IF bError THEN
	eCurrentState := E_MachineState.MACHINESTATE_Error;
	bBusy := FALSE;
	aPumps[nPumpNrRinsePump].M_Off();
	aPumps[nPumpNrWastePump].M_Off();
END_IF

//Prozessdaten aktualisieren
stProcessData.nObjId := nObjectID;
stProcessData.n32Data[0] := BOOL_TO_DINT(bIsInit);
stProcessData.n32Data[1] := eCurrentState;
stProcessData.n32Data[2] := stError.ErrorId;

stProcessData.n32Data[3] := BOOL_TO_DINT(bRinse);

stProcessData.n32Data[4] := BOOL_TO_DINT(aPumps[nPumpNrWastePump].P_bIsOn);
aObjProcData[nNotifyId] := stProcessData;

ACTION A_EmptyWaste:
IF nStateA_EmptyWaste = 0 THEN	//Wastepumpe einschalten
	aPumps[nPumpNrWastePump].M_On();
	tmrEmptyFluid(IN:= TRUE, PT:= T#10S);
	nStateA_EmptyWaste := 1;
ELSIF nStateA_EmptyWaste = 1 THEN //Warten auf Timer und Wastepumpe ausschalten
	tmrEmptyFluid();
	IF tmrEmptyFluid.Q THEN
		tmrEmptyFluid(IN:= FALSE);
		aPumps[nPumpNrWastePump].M_Off();
		IF NOT bLevelSensor THEN	//Leeren
			IF nPumpNrRinsePump > 0 THEN
				aPumps[nPumpNrRinsePump].M_Off();	
			END_IF
			stError.ErrorId := E_ErrorIdCmd.ERRORID_TimeOut;
			stError.POUState := nStateA_EmptyWaste;
			nStateA_EmptyWaste := 99;
		END_IF
		nStateA_EmptyWaste := 80;
	END_IF
ELSIF nStateA_EmptyWaste = 70 THEN
	tmrEmptyFluid(IN:= FALSE);
	nStateA_EmptyWaste := 80;
END_IF

//Errorhandling
IF nStateA_EmptyWaste = 99 THEN
	stError.Cmd := E_Action.ACTION_EmptyWaste;
	stError.POUAction := E_POUACT.POUACT_A_EmptyWaste;
	fbErrorList.M_Add(stError);
END_IF
END_ACTION

ACTION A_Rinse:
//Überwachung des Wastebottles
stError.ErrorId := M_CheckBottles();
IF stError.ErrorId > 0 THEN
	stError.POUState := nStateA_Rinse;
	nStateA_Rinse := 99;
END_IF

CASE nStateA_Rinse OF
	0:	IF bRinseOn THEN
			//WastePump EIN
			//RinsePump EIN
			aPumps[nPumpNrWastePump].M_On();
			aPumps[nPumpNrRinsePump].P_nStartSpeed := aStRinseChannels[nRinseChannel].nStartSpeed;
			aPumps[nPumpNrRinsePump].P_nRatedSpeed := aStRinseChannels[nRinseChannel].nRatedSpeed;
			aPumps[nPumpNrRinsePump].P_nDelay := aStRinseChannels[nRinseChannel].nStartTime;
			IF aStRinseChannels[nRinseChannel].nValveNr > 0 THEN
				aValves[aStRinseChannels[nRinseChannel].nValveNr].M_On(1);
			END_IF
			
			IF aPumps[nPumpNrRinsePump].M_On() THEN
				IF tmrRinse.PT > T#0MS THEN
					tmrRinse.IN := TRUE;
					nStateA_Rinse := 1;
				ELSE
					nStateA_Rinse := 1;
				END_IF
			END_IF
		ELSE
			bEmptyWaste := TRUE;
			M_RinsePumpOff();
			nStateA_Rinse := 80;
		END_IF

	1:	//Rinse aktiv (Überwachung des LevelSensors und des Rinse-Timers
		tmrRinse();
		IF bRinseOn THEN
			IF tmrRinse.Q THEN
				nStateA_Rinse := 3;
				RETURN;	
			END_IF
		
			IF NOT bLevelSensor THEN	//RinsePumpe für 2s "AUS" und dann wieder "EIN"
				M_RinsePumpOff();
				tmrRinsePause(IN:= TRUE, PT:= T#2S);
				nStateA_Rinse := 2;
			END_IF
		ELSE
			tmrRinsePause(IN:= FALSE);
			nStateA_Rinse := 3;
		END_IF
		
	2:	//Warten bis Timer abgelaufen
		IF bRinseOn THEN
			tmrRinse();
			IF tmrRinse.Q THEN
				tmrRinsePause(IN:= FALSE);
				//Hier sollte der Sensor spätestens wieder frei sein
				IF NOT bLevelSensor THEN
					stError.ErrorId := E_ErrorIdCmd.ERRORID_TimeOut;
					stError.POUState := nStateA_Rinse;
					nStateA_Rinse := 99; //Error
				ELSE
					nStateA_Rinse := 0; //Pumpe wieder einschalten??	
				END_IF
			END_IF
		ELSE
			tmrRinse(IN:= FALSE);
			nStateA_Rinse := 3;
		END_IF
		
	3:	//Aus
		tmrRinse(IN:=FALSE);
		IF NOT bKeepWastePumpOn THEN
			bEmptyWaste := TRUE;
		END_IF
		M_RinsePumpOff();
		nStateA_Rinse := 80;
		
	70:	//Abbrechen
		aPumps[nPumpNrWastePump].M_Off();
		M_RinsePumpOff();

		tmrRinse(IN:= FALSE);
		nStateA_Rinse := 80;

	90: //Error - Abbrechen
		aPumps[nPumpNrWastePump].M_Off();
		M_RinsePumpOff();
		tmrRinse(IN:= FALSE);
		tmrRinsePause(IN:= FALSE);
END_CASE

//Errorhandling
IF nStateA_Rinse = 99 THEN
	aPumps[nPumpNrWastePump].M_Off();
	M_RinsePumpOff();
	tmrRinse(IN:= FALSE);
	tmrRinsePause(IN:= FALSE);
	stError.Cmd := E_Action.ACTION_Rinse;
	stError.POUAction := E_POUACT.POUACT_A_Rinse;
	fbErrorList.M_Add(stError);
END_IF
END_ACTION

ACTION A_SwitchPump:
IF nStateA_SwitchPump = 0 THEN
	//Welche Pumpe soll geschalten werden?
	//0= Waste
	//>0 = RinseChannel
	IF nSwitchChannel = 0 THEN
		IF bSwitchOn THEN	//Waste-Pumpe einschalten
			//Falls EmptyWaste noch aktiv ist, dieses abbrechen, da EmptyWaste die Pumpe wieder abschaltet
			M_CancelAction(E_Action.ACTION_EmptyWaste);
			aPumps[nPumpNrWastePump].M_On();
		ELSE	//Ausschalten
			aPumps[nPumpNrWastePump].M_Off();
		END_IF
		nStateA_SwitchPump := 80;
	ELSIF nSwitchChannel > 0 THEN
		IF bSwitchOn THEN	//Einschalten
			aPumps[nPumpNrRinsePump].P_nStartSpeed := aStRinseChannels[nRinseChannel].nStartSpeed;
			aPumps[nPumpNrRinsePump].P_nRatedSpeed := aStRinseChannels[nRinseChannel].nRatedSpeed;
			aPumps[nPumpNrRinsePump].P_nDelay := aStRinseChannels[nRinseChannel].nStartTime;
			IF aStRinseChannels[nRinseChannel].nValveNr > 0 THEN
				aValves[aStRinseChannels[nRinseChannel].nValveNr].M_On(1);
			END_IF				
		ELSE	//Ausschalten
			M_RinsePumpOff();
		END_IF
			nStateA_SwitchPump := 80;
	END_IF
ELSIF nStateA_SwitchPump = 70 THEN
	aPumps[nPumpNrWastePump].M_Off();
	M_RinsePumpOff();
	nStateA_SwitchPump := 80;
END_IF
END_ACTION

METHOD FB_init : BOOL
VAR_INPUT
	bInitRetains : BOOL; // if TRUE, the retain variables are initialized (warm start / cold start)
	bInCopyCode : BOOL;  // if TRUE, the instance afterwards gets moved into the copy code (online change)
END_VAR
eObjectType := E_ObjectType.OBJECTTYPE_WashStation;
eObjectGroup := E_ObjectGroup.OBJECTGROUP_Target OR E_ObjectGroup.OBJECTGROUP_Device;
END_METHOD

METHOD M_ApplyPos : ERRORID
VAR_INPUT
	eTargetRef 		: E_TargetRef;
	nPointSlotNr	: UINT;
	stPos 			: ST_3DPoint;
	bXPos			: BOOL;
	bYPos			: BOOL;
	bZPos			: BOOL;	
END_VAR

VAR
	stAbsPos		: ST_3DPoint;
END_VAR
IF eTargetRef = E_TargetRef.TARGETREF_SpecPoint THEN
	stAbsPos := P_stAbsPosLB;
	IF bXPos THEN
		aStWashPoints[nPointSlotNr].X := stPos.X - stAbsPos.X;
	END_IF
	IF bYPos THEN
		aStWashPoints[nPointSlotNr].Y := stPos.Y - stAbsPos.Y;
	END_IF
	IF bZPos THEN
		aStWashPoints[nPointSlotNr].Z := stPos.Z - stAbsPos.Z;
	END_IF		
ELSE
	M_ApplyPos := SUPER^.M_ApplyPos(eTargetRef, nPointSlotNr, stPos,bXPos, bYPos, bZPos);	
END_IF
END_METHOD

METHOD M_CancelAction
VAR_INPUT
	eAction : E_Action;
END_VAR
CASE eAction OF
	E_Action.ACTION_Rinse:
		IF bRinse AND nStateA_Rinse < 70 THEN
			nStateA_Rinse := 70;
		END_IF
	E_Action.ACTION_SwitchPump:
		IF bSwitchPump AND nStateA_SwitchPump < 70 THEN
			nStateA_SwitchPump := 70;
		END_IF
	E_Action.ACTION_EmptyWaste:
		IF bEmptyWaste AND nStateA_EmptyWaste < 70 THEN
			nStateA_EmptyWaste := 70;
		END_IF
END_CASE
END_METHOD

METHOD M_CheckAction : ERRORID
VAR_INPUT
	refActionData 	: REFERENCE TO ST_ActionData;
	pCorrelObject	: POINTER TO FB_Object;
END_VAR
IF refActionData.eAction = E_Action.ACTION_TeachTarget THEN
	IF NOT DINT_TO_UINT(refActionData.aParams[1]) = E_TargetRef.TARGETREF_SpecPoint AND (refActionData.aParams[2] = 1 AND refActionData.aParams[2] = 2) THEN
		M_CheckAction := E_ErrorIdCmd.ERRORID_InvalidTargetPointRef;
	END_IF
ELSIF refActionData.eAction = E_Action.ACTION_WashTool THEN
	//SpecPoint prüfen
	IF NOT (refActionData.aParams[1] > 0 AND refActionData.aParams[1] <= nNoOfWashPoints) THEN
		M_CheckAction := E_ErrorIdCmd.ERRORID_InvalidTargetPointNr;
		RETURN;
	END_IF
	//Washmode prüfen
	IF NOT(refActionData.aParams[2] = E_WashMode.MODE_WashInside OR
		refActionData.aParams[2] = E_WashMode.MODE_WashOutside OR
		refActionData.aParams[2] = E_WashMode.MODE_WashInOutside OR
		refActionData.aParams[2] = E_WashMode.MODE_DryOutside) THEN
		M_CheckAction := E_ErrorIdCmd.ERRORID_InvalidWashMode;
		RETURN;
	END_IF
	//BottleState prüfen
	M_CheckAction := M_CheckBottles();
END_IF
END_METHOD

METHOD M_CheckBottles : ERRORID
VAR_INPUT
END_VAR
//Systemliquidbottle OK?
IF nSysLiquidBottle > 0 THEN
	IF NOT aSensSysLiquidBottle[nSysLiquidBottle] THEN //Leer
		M_CheckBottles := E_ErrorIdCmd.ERRORID_LiquidBottleEmpty;
		RETURN;
	END_IF
END_IF
//Wastebottle OK?
IF nWasteBottle > 0 THEN
	IF NOT aSensWasteBottle[nWasteBottle] THEN //Voll
		M_CheckBottles := E_ErrorIdCmd.ERRORID_WasteBottleFull;
		RETURN;
	END_IF
END_IF
END_METHOD

METHOD M_CheckProcDataType : BOOL
VAR_INPUT
	eProcDataType : E_ProcDataType;
END_VAR
END_METHOD

METHOD M_ExeAction : ERRORID
VAR_INPUT
	refActionData : REFERENCE TO ST_ActionData;	
END_VAR
IF refActionData.eAction = E_Action.ACTION_Init THEN
	bIsInit := TRUE;
	RETURN;
ELSIF refActionData.eAction = E_Action.ACTION_SwitchPump THEN
	IF NOT bSwitchPump THEN
		nSwitchChannel := DINT_TO_USINT(refActionData.aParams[1]);
		IF NOT(nSwitchChannel >= 0 AND nSwitchChannel <= nNoOfRinseChannels) THEN
			M_ExeAction := E_ErrorIdCmd.ERRORID_InvalidPumpNr;
			RETURN;			
		END_IF
		bSwitchOn := DINT_TO_BOOL(refActionData.aParams[2]);
		bSwitchPump := TRUE;
	ELSE
		RETURN;
	END_IF
	
ELSIF refActionData.eAction = E_Action.ACTION_EmptyWaste THEN
	IF NOT aSensWasteBottle[nWasteBottle] THEN
		M_ExeAction := E_ErrorIdCmd.ERRORID_WasteBottleFull;
		RETURN;
	END_IF
	IF NOT bEmptyWaste THEN
		bEmptyWaste := TRUE;
	ELSE
		RETURN;
	END_IF

ELSIF refActionData.eAction = E_Action.ACTION_Stop THEN
	IF bRinse THEN
		bRinseOn := FALSE;
	ELSE
		aPumps[nPumpNrWastePump].M_Off();
		M_RinsePumpOff();
	END_IF	
	
ELSIF refActionData.eAction = E_Action.ACTION_Rinse THEN
	nRinseChannel := DINT_TO_USINT(refActionData.aParams[1]);
	tmrRinse.PT := DINT_TO_TIME(refActionData.aParams[3]);
	IF NOT(nRinseChannel >= 1 AND nRinseChannel <= nNoOfRinseChannels) THEN
		M_ExeAction := E_ErrorIdCmd.ERRORID_InvalidRinseChannel;
		RETURN;
	END_IF
	nPumpNrRinsePump := aStRinseChannels[nRinseChannel].nPumpNr;
	bRinseOn := DINT_TO_BOOL(refActionData.aParams[2]);
	bKeepWastePumpOn := DINT_TO_BOOL(refActionData.aParams[4]);
	bRinse := TRUE;
ELSE
	M_ExeAction := E_ErrorIdCmd.ERRORID_InvalidAction;
	RETURN;
END_IF
bBusy := TRUE;
eCurrentState:= E_MachineState.MACHINESTATE_Active;
END_METHOD

METHOD M_GetAbsPos : ST_3DPoint
VAR_INPUT
	pChildPos	: POINTER TO ST_3DPoint;
	eTargetRef 	: E_TargetRef;
	nParam1		: UINT;
 	nParam2		: UINT;
	nParam3		: USINT;
	nParam4		: USINT;
	nZLevel		: USINT;
END_VAR
VAR_OUTPUT
	nErrorId 	: ERRORID;
	lrAngle		: LREAL;
END_VAR
VAR
	stLocPosLB : ST_3DPoint;
END_VAR
IF eTargetRef = E_TargetRef.TARGETREF_SpecPoint THEN
	IF nParam1 > 0 AND nParam1 <= cMaxWashPoints THEN
		stLocPosLB := P_stRelPosLB;
		stLocPosLB := F_Add3DPoints(stLocPosLB,aStWashPoints[nParam1]);
		M_GetAbsPos := pParentTarget^.M_GetAbsPos(pChildPos := ADR(stLocPosLB), eTargetRef:= E_TargetRef.TARGETREF_LeftBottom,
														nParam1:= 0,
														nParam2:= 0, nParam3:= 0,nParam4:= 0, nZLevel:= 0,
														lrAngle => lrAngle, nErrorId=> nErrorId);		
	ELSE
		nErrorId := E_ErrorIdCmd.ERRORID_InvalidTargetPointNr;
	END_IF
ELSE
	M_GetAbsPos := SUPER^.M_GetAbsPos(pChildPos := pChildPos, eTargetRef:= eTargetRef,
													nParam1:= nParam1,
													nParam2:= nParam2, nParam3:= nParam3, nParam4:= 0, nZLevel:= nZLevel,
													lrAngle => lrAngle, nErrorId=> nErrorId);	
END_IF
END_METHOD

METHOD M_GetActionBusy : BOOL
VAR_INPUT
	eAction : E_Action;
END_VAR
IF eAction = E_Action.ACTION_SwitchPump THEN
	M_GetActionBusy := bSwitchPump;
ELSIF eAction = E_Action.ACTION_EmptyWaste THEN
	M_GetActionBusy := bEmptyWaste;
ELSIF eAction = E_Action.ACTION_Rinse THEN
	M_GetActionBusy := bRinse;
END_IF
END_METHOD

METHOD M_GetAllProps : ERRORID
VAR_INPUT
	refCmdData : REFERENCE TO  ST_CmdData;
END_VAR

VAR
	i : USINT;
END_VAR
SUPER^.M_GetAllProps(refCmdData); 

//RinseChannels
nCurrentPropIndex := nCurrentPropIndex + 1;
refCmdData.n32Data[nCurrentPropIndex] := nNoOfRinseChannels;
//In Abhängigkeit von der Anzahl der RinseChannels , diese aus RinseChannel-Array lesen
FOR i:= 1 TO nNoOfRinseChannels BY 1 DO
	nCurrentPropIndex := nCurrentPropIndex + 1;	//PumpNr
	refCmdData.n32Data[nCurrentPropIndex] := aStRinseChannels[i].nPumpNr;
	nCurrentPropIndex := nCurrentPropIndex + 1;	//ValveNr
	refCmdData.n32Data[nCurrentPropIndex] := aStRinseChannels[i].nValveNr;
	nCurrentPropIndex := nCurrentPropIndex + 1;	//StartSpeed in %
	refCmdData.n32Data[nCurrentPropIndex] := aStRinseChannels[i].nStartSpeed;
	nCurrentPropIndex := nCurrentPropIndex + 1;	//RatedSpeed in %
	refCmdData.n32Data[nCurrentPropIndex] := aStRinseChannels[i].nRatedSpeed;
	nCurrentPropIndex := nCurrentPropIndex + 1;	//StartTime in ms
	refCmdData.n32Data[nCurrentPropIndex] := aStRinseChannels[i].nStartTime;
END_FOR

//WashPoints
nCurrentPropIndex := nCurrentPropIndex + 1;
refCmdData.n32Data[nCurrentPropIndex] := nNoOfWashPoints; 
//In Abhängigkeit von der Anzahl der Waschpunkte , diese aus WashPoint-Array lesen
FOR i:= 1 TO nNoOfWashPoints BY 1 DO
	nCurrentPropIndex := nCurrentPropIndex + 1;
	refCmdData.n32Data[nCurrentPropIndex] := REAL_TO_DINT(aStWashPoints[i].X);
	nCurrentPropIndex := nCurrentPropIndex + 1;
	refCmdData.n32Data[nCurrentPropIndex] := REAL_TO_DINT(aStWashPoints[i].Y);
	nCurrentPropIndex := nCurrentPropIndex + 1;
	refCmdData.n32Data[nCurrentPropIndex] := REAL_TO_DINT(aStWashPoints[i].Z);
	nCurrentPropIndex := nCurrentPropIndex + 1;
	refCmdData.n32Data[nCurrentPropIndex] := REAL_TO_DINT(aStWashPoints[i].nRinseChannel);
END_FOR

nCurrentPropIndex := nCurrentPropIndex + 1;
refCmdData.n32Data[nCurrentPropIndex] := nPumpNrWastePump;
nCurrentPropIndex := nCurrentPropIndex + 1;
refCmdData.n32Data[nCurrentPropIndex] := nSysLiquidBottle;
nCurrentPropIndex := nCurrentPropIndex + 1;
refCmdData.n32Data[nCurrentPropIndex] := nWasteBottle;
nCurrentPropIndex := nCurrentPropIndex + 1;
refCmdData.n32Data[nCurrentPropIndex] := nValveNrAirShower;
nCurrentPropIndex := nCurrentPropIndex + 1;
refCmdData.n32Data[nCurrentPropIndex] := nGCodeTargetNr;
END_METHOD

METHOD M_GetProcData : DINT
VAR_INPUT
	eProcDataType : E_ProcDataType;
END_VAR
END_METHOD

METHOD M_GetRinseChannel : USINT
VAR_INPUT
	nWashPointNr : USINT;
END_VAR
IF nWashPointNr > 0 AND nWashPointNr <= nNoOfWashPoints THEN
	M_GetRinseChannel := aStWashPoints[nWashPointNr].nRinseChannel;
END_IF
END_METHOD

METHOD M_Reset
bError := FALSE;
bBusy := FALSE;
eCurrentState := E_MachineState.MACHINESTATE_Idle;
END_METHOD

METHOD PRIVATE M_RinsePumpOff
VAR_INPUT
END_VAR

VAR
	i		: USINT;
	nTemp 	: USINT;
END_VAR
FOR i := 1 TO nNoOfRinseChannels BY 1 DO
	nTemp := aStRinseChannels[i].nPumpNr;
	IF nTemp > 0 THEN
		aPumps[nTemp].M_Off();
	END_IF
	nTemp := aStRinseChannels[i].nValveNr;
	IF nTemp > 0 THEN
		aValves[nTemp].M_Off();
	END_IF
END_FOR
END_METHOD

METHOD M_SetAllProps : ERRORID
VAR_INPUT
	refCmdData : REFERENCE TO  ST_CmdData;
END_VAR

VAR
	i : USINT;
END_VAR
M_SetAllProps := SUPER^.M_SetAllProps(refCmdData);

IF M_SetAllProps > 0 THEN
	RETURN;
END_IF

//RinseChannels
nCurrentPropIndex := nCurrentPropIndex + 1;
nSpecPropIndex := nCurrentPropIndex;
nNoOfRinseChannels := DINT_TO_USINT(refCmdData.n32Data[nCurrentPropIndex]); 
//In Abhängigkeit von der Anzahl der RinseChannels , diese in RinseChannel-Array schreiben
IF NOT (nNoOfRinseChannels > 0 AND nNoOfRinseChannels <= cMaxRinseChannels) THEN
	M_SetAllProps := E_ErrorIdObjMgmt.ERRORID_InvalidNoOfRinseChannels;
	RETURN;
END_IF

FOR i:= 1 TO nNoOfRinseChannels BY 1 DO
	nCurrentPropIndex := nCurrentPropIndex + 1; //PumpNr
	IF refCmdData.n32Data[nCurrentPropIndex] >= 0 AND refCmdData.n32Data[nCurrentPropIndex] <= cNoOfPumps THEN
		aStRinseChannels[i].nPumpNr := DINT_TO_USINT(refCmdData.n32Data[nCurrentPropIndex]);
	ELSE
		M_SetAllProps := E_ErrorIdCmd.ERRORID_InvalidPumpNr;
		RETURN;
	END_IF
	nCurrentPropIndex := nCurrentPropIndex + 1;	//ValveNr
	IF refCmdData.n32Data[nCurrentPropIndex] >= 0 AND refCmdData.n32Data[nCurrentPropIndex] <= cNoOfValves THEN
		aStRinseChannels[i].nValveNr := DINT_TO_USINT(refCmdData.n32Data[nCurrentPropIndex]);
	ELSE
		M_SetAllProps := E_ErrorIdObjMgmt.ERRORID_InvalidValveNumber;
		RETURN;
	END_IF
	nCurrentPropIndex := nCurrentPropIndex + 1;	//StartSpeed in %
	aStRinseChannels[i].nStartSpeed := DINT_TO_USINT(refCmdData.n32Data[nCurrentPropIndex]);
	nCurrentPropIndex := nCurrentPropIndex + 1;	//RatedSpeed in %
	aStRinseChannels[i].nRatedSpeed := DINT_TO_USINT(refCmdData.n32Data[nCurrentPropIndex]);
	nCurrentPropIndex := nCurrentPropIndex + 1;	//StartTime in ms
	aStRinseChannels[i].nStartTime := DINT_TO_UINT(refCmdData.n32Data[nCurrentPropIndex]);
END_FOR

//WashPoints
nCurrentPropIndex := nCurrentPropIndex + 1;
nNoOfWashPoints := DINT_TO_USINT(refCmdData.n32Data[nCurrentPropIndex]); 
//In Abhängigkeit von der Anzahl der Waschpunkte , diese in WashPoint-Array schreiben
IF NOT (nNoOfWashPoints > 0 AND nNoOfWashPoints <= cMaxWashPoints) THEN
	M_SetAllProps := E_ErrorIdObjMgmt.ERRORID_InvalidNoOfSpecPoints;
	RETURN;
END_IF

FOR i:= 1 TO nNoOfWashPoints BY 1 DO
	nCurrentPropIndex := nCurrentPropIndex + 1;
	aStWashPoints[i].X := DINT_TO_REAL(refCmdData.n32Data[nCurrentPropIndex]);
	nCurrentPropIndex := nCurrentPropIndex + 1;
	aStWashPoints[i].Y := DINT_TO_REAL(refCmdData.n32Data[nCurrentPropIndex]);
	nCurrentPropIndex := nCurrentPropIndex + 1;
	aStWashPoints[i].Z := DINT_TO_REAL(refCmdData.n32Data[nCurrentPropIndex]);
	nCurrentPropIndex := nCurrentPropIndex + 1;
	//Zugeordneter RinseChannel
	aStWashPoints[i].nRinseChannel := DINT_TO_USINT(refCmdData.n32Data[nCurrentPropIndex]);;
END_FOR

//WastePump
nCurrentPropIndex := nCurrentPropIndex + 1;
IF refCmdData.n32Data[nCurrentPropIndex] >= 1 AND refCmdData.n32Data[nCurrentPropIndex] <= cNoOfPumps THEN
	nPumpNrWastePump := DINT_TO_USINT(refCmdData.n32Data[nCurrentPropIndex]);
ELSE
	M_SetAllProps := E_ErrorIdCmd.ERRORID_InvalidPumpNr;
END_IF

//LiquidBottle
nCurrentPropIndex := nCurrentPropIndex + 1;
IF refCmdData.n32Data[nCurrentPropIndex] >= 1 AND refCmdData.n32Data[nCurrentPropIndex] <= cNoOfLiquidBottles THEN
	nSysLiquidBottle := DINT_TO_USINT(refCmdData.n32Data[nCurrentPropIndex]);
ELSE
	M_SetAllProps := E_ErrorIdObjMgmt.ERRORID_InvalidLiquidbottle;
END_IF

//WasteBottle
nCurrentPropIndex := nCurrentPropIndex + 1;
IF refCmdData.n32Data[nCurrentPropIndex] >= 1 AND refCmdData.n32Data[nCurrentPropIndex] <= cNoOfWasteBottles THEN
	nWasteBottle := DINT_TO_USINT(refCmdData.n32Data[nCurrentPropIndex]);
ELSE
	M_SetAllProps := E_ErrorIdObjMgmt.ERRORID_InvalidWastebottle;
END_IF

//ValveNrDrying (Trockendusche für pH Elektrode)
nCurrentPropIndex := nCurrentPropIndex + 1;
IF refCmdData.n32Data[nCurrentPropIndex] >= 0 AND refCmdData.n32Data[nCurrentPropIndex] <= cNoOfValves THEN
	nValveNrAirShower := DINT_TO_USINT(refCmdData.n32Data[nCurrentPropIndex]);
ELSE
	M_SetAllProps := E_ErrorIdObjMgmt.ERRORID_InvalidValveNumber;
END_IF
nCurrentPropIndex := nCurrentPropIndex + 1;
nGCodeTargetNr := DINT_TO_UINT(refCmdData.n32Data[nCurrentPropIndex]);
nNoOfProps := nCurrentPropIndex + 1;
END_METHOD

METHOD M_SetSingleProp : ERRORID
VAR_INPUT
	refCmdData : REFERENCE TO  ST_CmdData;
END_VAR

VAR
	i : UINT;
	nIndex					: UINT;
	nIndexRinseChannels	 	: UINT;
	nIndexWashPoints 	 	: UINT;
	nIndexRestProps 	 	: UINT;
END_VAR
nIndexRinseChannels := nSpecPropIndex;
nIndexWashPoints := nIndexRinseChannels + nNoOfRinseChannels * 5 + 1;
nIndexRestProps := nIndexWashPoints + nNoOfWashPoints * 4 + 1;

//Section: RinseChannels
IF refCmdData.aHeader[1] > nIndexRinseChannels AND refCmdData.aHeader[1] < nIndexWashPoints THEN
	FOR i:= 1 TO nNoOfRinseChannels BY 1 DO
		//ersten Index innerhalb der Section ermitteln
		nIndex := nIndexRinseChannels + ((i - 1) * 5) + 1;
		IF refCmdData.aHeader[1] = nIndex THEN	//PumpNr
			IF refCmdData.n32Data[0] >= 0 AND refCmdData.n32Data[0] <= cNoOfPumps THEN
				aStRinseChannels[i].nPumpNr := DINT_TO_USINT(refCmdData.n32Data[0]);
			ELSE
				M_SetSingleProp := E_ErrorIdCmd.ERRORID_InvalidPumpNr;
				RETURN;
			END_IF
			RETURN;
		ELSIF refCmdData.aHeader[1] = nIndex + 1 THEN	//ValveNr
			IF refCmdData.n32Data[0] >= 0 AND refCmdData.n32Data[0] <= cNoOfValves THEN
				aStRinseChannels[i].nValveNr := DINT_TO_USINT(refCmdData.n32Data[0]);
			ELSE
				M_SetSingleProp := E_ErrorIdObjMgmt.ERRORID_InvalidValveNumber;
				RETURN;
			END_IF
		ELSIF refCmdData.aHeader[1] = nIndex + 2 THEN	//StartSpeed in %
			aStRinseChannels[i].nStartSpeed := DINT_TO_USINT(refCmdData.n32Data[0]);	
		ELSIF refCmdData.aHeader[1] = nIndex + 3 THEN	//RatedSpeed in %
			aStRinseChannels[i].nRatedSpeed := DINT_TO_USINT(refCmdData.n32Data[0]);
		ELSIF refCmdData.aHeader[1] = nIndex + 4 THEN	//StartTime in ms
			aStRinseChannels[i].nStartTime := DINT_TO_UINT(refCmdData.n32Data[0]);
		END_IF		
	END_FOR
//Section: Washpoints	
ELSIF refCmdData.aHeader[1] > nIndexWashPoints AND refCmdData.aHeader[1] < nIndexRestProps THEN
	FOR i:= 1 TO nNoOfWashPoints BY 1 DO
		//ersten Index innerhalb der Section ermitteln
		nIndex := nIndexWashPoints + ((i - 1) * 4) + 1;
		IF refCmdData.aHeader[1] = nIndex THEN
			aStWashPoints[i].X := DINT_TO_REAL(refCmdData.n32Data[0]);
		ELSIF refCmdData.aHeader[1] = nIndex + 1 THEN
			aStWashPoints[i].Y := DINT_TO_REAL(refCmdData.n32Data[0]);
		ELSIF refCmdData.aHeader[1] = nIndex + 2 THEN
			aStWashPoints[i].Z := DINT_TO_REAL(refCmdData.n32Data[0]);
		ELSIF refCmdData.aHeader[1] = nIndex + 3 THEN
			M_SetSingleProp := E_ErrorIdCmd.ERRORID_InvalidProperty;
		END_IF			
	END_FOR
//Restliche Props
ELSIF refCmdData.aHeader[1] >= nIndexRestProps AND refCmdData.aHeader[1] < nNoOfProps THEN
	CASE (refCmdData.aHeader[1] - nIndexRestProps) OF
		0: //PumpNrWaste
			IF refCmdData.n32Data[0] > 0 AND refCmdData.n32Data[0] <= cNoOfPumps THEN
				nPumpNrWastePump := DINT_TO_USINT(refCmdData.n32Data[0]);
			ELSE
				M_SetSingleProp := E_ErrorIdCmd.ERRORID_InvalidPumpNr;
			END_IF			
		1: //LiquidBottle
			IF refCmdData.n32Data[0] > 0 AND refCmdData.n32Data[0] <= cNoOfLiquidBottles THEN
				nSysLiquidBottle := DINT_TO_USINT(refCmdData.n32Data[0]);
			ELSE
				M_SetSingleProp := E_ErrorIdObjMgmt.ERRORID_InvalidLiquidbottle;
			END_IF			
		2: //WasteBottle
			IF refCmdData.n32Data[0] > 0 AND refCmdData.n32Data[0] <= cNoOfWasteBottles THEN
				nWasteBottle := DINT_TO_USINT(refCmdData.n32Data[0]);
			ELSE
				M_SetSingleProp := E_ErrorIdObjMgmt.ERRORID_InvalidWastebottle;
			END_IF
		3: //ValveNrDrying (Trockendusche für pH Elektrode)
			IF refCmdData.n32Data[0] >= 0 AND refCmdData.n32Data[0] <= cNoOfValves THEN
				nValveNrAirShower := DINT_TO_USINT(refCmdData.n32Data[0]);
			ELSE
				M_SetSingleProp := E_ErrorIdObjMgmt.ERRORID_InvalidValveNumber;
			END_IF			
	END_CASE	
ELSE
	M_SetSingleProp := SUPER^.M_SetSingleProp(refCmdData);
END_IF
END_METHOD

METHOD M_Stop : ERRORID
VAR_INPUT
END_VAR
IF bRinse AND nStateA_Rinse < 70 THEN
	nStateA_Rinse := 70;
END_IF

IF bSwitchPump AND nStateA_SwitchPump < 70 THEN
	nStateA_SwitchPump := 70;
END_IF

aPumps[nPumpNrWastePump].M_Off();

M_SwitchAirShower(FALSE);

(*IF bEmptyFluid AND nStateA_EmptyFluid < 70 THEN
	nStateA_EmptyFluid := 70;
END_IF*)
END_METHOD

METHOD M_SwitchAirShower : ERRORID
VAR_INPUT
	bOn	: BOOL;
END_VAR
IF bOn THEN
	IF nValveNrAirShower > 0 THEN
		aValves[nValveNrAirShower].M_On(1);
	ELSE
		M_SwitchAirShower := E_ErrorIdCmd.ERRORID_WashStationHasNoAirShower;
	END_IF
ELSE
	IF nValveNrAirShower > 0 THEN
		aValves[nValveNrAirShower].M_Off();
	END_IF
END_IF
END_METHOD

PROPERTY P_nGCodeTargetNr : UINT
GET
P_nGCodeTargetNr := nGCodeTargetNr;
END_GET
END_PROPERTY

END_FUNCTION_BLOCK

// ---- Objects/Targets/Active/FB_TipCalibrator.TcPOU
FUNCTION_BLOCK FB_TipCalibrator EXTENDS FB_ActiveTarget
VAR_INPUT
END_VAR

VAR
	bNumberOfSpecPoints	: USINT;
	stPassIntersectPoint: ST_3DPoint;
	stCalibPoint		: ST_3DPoint;
	bLegacy				: BOOL;	
END_VAR

//Prozessdaten aktualisieren
stProcessData.nObjId := nObjectID;
stProcessData.n32Data[0] := BOOL_TO_DINT(bIsInit);
stProcessData.n32Data[1] := E_MachineState.MACHINESTATE_Idle;
stProcessData.n32Data[2] := 0;
stProcessData.n32Data[3] := BOOL_TO_DINT(P_bXSensor);
stProcessData.n32Data[4] := BOOL_TO_DINT(P_bYSensor); 

aObjProcData[nNotifyId] := stProcessData;

METHOD FB_init : BOOL
VAR_INPUT
	bInitRetains : BOOL; // if TRUE, the retain variables are initialized (warm start / cold start)
	bInCopyCode : BOOL;  // if TRUE, the instance afterwards gets moved into the copy code (online change)
END_VAR
eObjectType := E_ObjectType.OBJECTTYPE_TipCalibrator;
eObjectGroup := E_ObjectGroup.OBJECTGROUP_Target OR E_ObjectGroup.OBJECTGROUP_Device;
END_METHOD

METHOD M_CancelAction
VAR_INPUT
	eAction : E_Action;
END_VAR
END_METHOD

METHOD M_CheckAction : ERRORID
VAR_INPUT
	refActionData 	: REFERENCE TO ST_ActionData;
	pCorrelObject	: POINTER TO FB_Object;
END_VAR
IF refActionData.eAction <> E_Action.ACTION_MoveToTarget THEN
	M_CheckAction := 8989;	
END_IF
END_METHOD

METHOD M_CheckProcDataType : BOOL
VAR_INPUT
	eProcDataType : E_ProcDataType;
END_VAR
END_METHOD

METHOD M_ExeAction : ERRORID
VAR_INPUT
	refActionData : REFERENCE TO ST_ActionData;	
END_VAR
IF refActionData.eAction = E_Action.ACTION_Init THEN
	bIsInit := TRUE;
END_IF
END_METHOD

METHOD M_GetAbsPos : ST_3DPoint
VAR_INPUT
	pChildPos	: POINTER TO ST_3DPoint;
	eTargetRef 	: E_TargetRef;
	nParam1		: UINT;
 	nParam2		: UINT;
	nParam3		: USINT;
	nParam4		: USINT;
	nZLevel		: USINT;
END_VAR
VAR_OUTPUT
	nErrorId 	: ERRORID;
	lrAngle		: LREAL;
END_VAR
VAR
	stLocPosLB : ST_3DPoint;
END_VAR
IF eTargetRef = E_TargetRef.TARGETREF_SpecPoint THEN
	stLocPosLB := P_stRelPosLB;
	IF nParam1 = 1 THEN
		stLocPosLB := F_Add3DPoints(stLocPosLB,stPassIntersectPoint);
	ELSIF nParam1 = 2 THEN
		stLocPosLB := F_Add3DPoints(stLocPosLB,stCalibPoint);
	ELSE
		nErrorId := E_ErrorIdCmd.ERRORID_InvalidTargetPointNr;
		RETURN;
	END_IF
	M_GetAbsPos := pParentTarget^.M_GetAbsPos(pChildPos := ADR(stLocPosLB), eTargetRef:= E_TargetRef.TARGETREF_LeftBottom,
												nParam1:= 0,
												nParam2:= 0, nParam3:= 0, nParam4:= 0,nZLevel:= 0,
												lrAngle => lrAngle, nErrorId=> nErrorId);
ELSE
	M_GetAbsPos := SUPER^.M_GetAbsPos(pChildPos := pChildPos, eTargetRef:= eTargetRef,
													nParam1:= nParam1,
													nParam2:= nParam2, nParam3:= nParam3, nParam4:= 0, nZLevel:= nZLevel,
													lrAngle => lrAngle, nErrorId=> nErrorId);	
END_IF
END_METHOD

METHOD M_GetActionBusy : BOOL
VAR_INPUT
	eAction : E_Action;
END_VAR
END_METHOD

METHOD M_GetAllProps : ERRORID
VAR_INPUT
	refCmdData : REFERENCE TO  ST_CmdData;
END_VAR
SUPER^.M_GetAllProps(refCmdData);

nCurrentPropIndex := nCurrentPropIndex + 1;
refCmdData.n32Data[nCurrentPropIndex] := bNumberOfSpecPoints;
nCurrentPropIndex := nCurrentPropIndex + 1;
refCmdData.n32Data[nCurrentPropIndex] := REAL_TO_DINT(stPassIntersectPoint.X);
nCurrentPropIndex := nCurrentPropIndex + 1;
refCmdData.n32Data[nCurrentPropIndex] := REAL_TO_DINT(stPassIntersectPoint.Y);
nCurrentPropIndex := nCurrentPropIndex + 1;
refCmdData.n32Data[nCurrentPropIndex] := REAL_TO_DINT(stPassIntersectPoint.Z);
nCurrentPropIndex := nCurrentPropIndex + 1;
refCmdData.n32Data[nCurrentPropIndex] := REAL_TO_DINT(stCalibPoint.X);
nCurrentPropIndex := nCurrentPropIndex + 1;
refCmdData.n32Data[nCurrentPropIndex] := REAL_TO_DINT(stCalibPoint.Y);
nCurrentPropIndex := nCurrentPropIndex + 1;
refCmdData.n32Data[nCurrentPropIndex] := REAL_TO_DINT(stCalibPoint.Z);
nCurrentPropIndex := nCurrentPropIndex + 1;
refCmdData.n32Data[nCurrentPropIndex] := BOOL_TO_DINT(bLegacy);
END_METHOD

METHOD M_GetProcData : DINT
VAR_INPUT
	eProcDataType : E_ProcDataType;
END_VAR
END_METHOD

METHOD M_SetAllProps : ERRORID
VAR_INPUT
	refCmdData : REFERENCE TO  ST_CmdData;
END_VAR
M_SetAllProps := SUPER^.M_SetAllProps(refCmdData);

IF M_SetAllProps > 0 THEN
	RETURN;
END_IF

nCurrentPropIndex := nCurrentPropIndex + 1;
nSpecPropIndex := nCurrentPropIndex;
bNumberOfSpecPoints := DINT_TO_USINT(refCmdData.n32Data[nCurrentPropIndex]);
IF bNumberOfSpecPoints <> 2 THEN
	M_SetAllProps := E_ErrorIdObjMgmt.ERRORID_InvalidNoOfSpecPoints;
	RETURN;
END_IF
nCurrentPropIndex := nCurrentPropIndex + 1;
stPassIntersectPoint.X := DINT_TO_REAL(refCmdData.n32Data[nCurrentPropIndex]);
nCurrentPropIndex := nCurrentPropIndex + 1; 
stPassIntersectPoint.Y := DINT_TO_REAL(refCmdData.n32Data[nCurrentPropIndex]);
nCurrentPropIndex := nCurrentPropIndex + 1;
stPassIntersectPoint.Z := DINT_TO_REAL(refCmdData.n32Data[nCurrentPropIndex]);
nCurrentPropIndex := nCurrentPropIndex + 1;
stCalibPoint.X := DINT_TO_REAL(refCmdData.n32Data[nCurrentPropIndex]);
nCurrentPropIndex := nCurrentPropIndex + 1;
stCalibPoint.Y := DINT_TO_REAL(refCmdData.n32Data[nCurrentPropIndex]);
nCurrentPropIndex := nCurrentPropIndex + 1;
stCalibPoint.Z := DINT_TO_REAL(refCmdData.n32Data[nCurrentPropIndex]);
nCurrentPropIndex := nCurrentPropIndex + 1;
bLegacy := DINT_TO_BOOL(refCmdData.n32Data[nCurrentPropIndex]);
nNoOfProps := nCurrentPropIndex + 1;
END_METHOD

METHOD M_SetSingleProp : ERRORID
VAR_INPUT
	refCmdData : REFERENCE TO  ST_CmdData;
END_VAR
IF nSpecPropIndex = refCmdData.aHeader[1] THEN
	M_SetSingleProp := E_ErrorIdCmd.ERRORID_InvalidProperty; //Anzahl Specpoints darf nicht verändert werden
ELSIF (nSpecPropIndex + 1) = refCmdData.aHeader[1] THEN
	stPassIntersectPoint.X := DINT_TO_REAL(refCmdData.n32Data[0]);
ELSIF (nSpecPropIndex + 2) = refCmdData.aHeader[1] THEN
	stPassIntersectPoint.Y := DINT_TO_REAL(refCmdData.n32Data[0]);
ELSIF (nSpecPropIndex + 3) = refCmdData.aHeader[1] THEN
	stPassIntersectPoint.Z := DINT_TO_REAL(refCmdData.n32Data[0]);
ELSIF (nSpecPropIndex + 4) = refCmdData.aHeader[1] THEN
	stCalibPoint.X := DINT_TO_REAL(refCmdData.n32Data[0]);
ELSIF (nSpecPropIndex + 5) = refCmdData.aHeader[1] THEN
	stCalibPoint.Y := DINT_TO_REAL(refCmdData.n32Data[0]);
ELSIF (nSpecPropIndex + 6) = refCmdData.aHeader[1] THEN
	stCalibPoint.Z := DINT_TO_REAL(refCmdData.n32Data[0]);
ELSE
	M_SetSingleProp := SUPER^.M_SetSingleProp(refCmdData);
END_IF
END_METHOD

METHOD M_Stop : ERRORID
VAR_INPUT
END_VAR
END_METHOD

PROPERTY P_bLegacy : BOOL
GET
P_bLegacy := bLegacy;
END_GET
END_PROPERTY

PROPERTY P_bXSensor : BOOL
GET
P_bXSensor := stTipCalibrator.bXSensor XOR stTipCalibrator.bInvert;
END_GET
END_PROPERTY

PROPERTY P_bYSensor : BOOL
GET
P_bYSensor := stTipCalibrator.bYSensor XOR stTipCalibrator.bInvert;
END_GET
END_PROPERTY

PROPERTY P_stCalibPoint : ST_3DPoint
GET
P_stCalibPoint := stCalibPoint;
END_GET
SET
stCalibPoint := P_stCalibPoint;
END_SET
END_PROPERTY

END_FUNCTION_BLOCK

// ---- Objects/Targets/Active/FB_Stroboscope.TcPOU
FUNCTION_BLOCK FB_Stroboscope EXTENDS FB_WorkplateCamera
VAR_INPUT
END_VAR
VAR
	nMultiZNr				: USINT;
	nCamDelay				: UINT;
	nStrobDelay				: UINT;
	nStrobDelay2			: UINT;
	aDroplist				: ARRAY[1..16] OF USINT;
	
	fbSdoWrite	: FB_SDO_WRITE;

	bNewCamDelay			: BOOL;
	bSendCamDelay			: BOOL;
	bSendCamDelayFlag		: BOOL := TRUE;
	
	bNewStrobDelay			: BOOL;
	bSendStrobDelay			: BOOL;
	bSendStrobDelayFlag		: BOOL := TRUE;

	bNewStrobDelay2			: BOOL;
	bSendStrobDelay2		: BOOL;
	bSendStrobDelay2Flag	: BOOL := TRUE;

	bNewDropList1_4			: BOOL;
	bSendDroplist1_4		: BOOL;
	bSendDroplist1_4Flag	: BOOL := TRUE;

	bNewDropList5_8			: BOOL;
	bSendDroplist5_8		: BOOL;
	bSendDroplist5_8Flag	: BOOL := TRUE;

	bNewDropList9_12		: BOOL;
	bSendDroplist9_12		: BOOL;
	bSendDroplist9_12Flag	: BOOL := TRUE;

	bNewDropList13_16		: BOOL;
	bSendDroplist13_16		: BOOL;
	bSendDroplist13_16Flag	: BOOL := TRUE;
	
	bSendStrobTestFlag		: BOOL := TRUE;
	pFbMultiZ				: POINTER TO FB_MultiZRef;
	
	nGCodeTargetNr	: UINT;
	
	//****************************************Aktionvariablen****************************************************
	
	//Action: "StrobTest"	(das Stroboskop mit 125 triggern (zu Testzwecken))
	bStrobTest			: BOOL;
	nStateA_StrobTest	: USINT;
	bStrobTestCtrl		: BOOL;
	
	nSendPauseCnt		: USINT;
END_VAR

IF bInitFB THEN
	bInitFB := FALSE;
	//Fehlerstruktur vorausfüllen
	stError.ObjectId := nObjectID;
	stError.HardwareGrp := E_HardwareGrp.Nothing;
	stError.POU := E_POU.POU_FB_Stroboscope;
END_IF

CASE eCurrentState OF
	E_MachineState.MACHINESTATE_Active:
	IF bStrobTest THEN
		A_StrobTest();
		IF nStateA_StrobTest = 80 THEN
			bStrobTest := FALSE;
			nStateA_StrobTest := 0;
			eCurrentState := E_MachineState.MACHINESTATE_Ready;
		ELSIF nStateA_StrobTest = 99 THEN
			bStrobTest := FALSE;
			nStateA_StrobTest := 0;
			stError.Cmd := E_Action.ACTION_StrobTest;
			fbErrorList.M_Add(stError);	//Error in Error-Liste eintragen
			eCurrentState := E_MachineState.MACHINESTATE_Error;
		END_IF
	END_IF
	
	E_MachineState.MACHINESTATE_Ready:
		bBusy := FALSE;
		eCurrentState := E_MachineState.MACHINESTATE_Idle;
	
	E_MachineState.MACHINESTATE_Error:
		bBusy := FALSE;
END_CASE

IF nSendPauseCnt < 100 THEN
	nSendPauseCnt := nSendPauseCnt + 1;
ELSE
	IF bSendCamDelay THEN
		IF bSendCamDelayFlag XOR fbSdoWrite.bBusy THEN
			bSendCamDelayFlag := FALSE;
			pFbMultiZ^.stStrobTrigger.nCamDelay := nCamDelay;
			fbSdoWrite(sADSNetID:= pFbMultiZ^.P_sAdsNetId, nPortNr:= pFbMultiZ^.P_nAdsPort,
						nIndex:= cPiezoCamDelay.nIndex, nSubIndex:= cPiezoCamDelay.nSubIndex, 
						nDataLength:= cPiezoCamDelay.nLength, nData:= pFbMultiZ^.stStrobTrigger.nCamDelay, bExecute:= TRUE);		
		END_IF
		
		IF NOT fbSdoWrite.bBusy THEN
			nSendPauseCnt := 0;
			bSendCamDelayFlag := TRUE;
			bSendCamDelay := FALSE;
			IF fbSdoWrite.bError THEN
				stError.Cmd := 0;
				fbSdoWrite(bExecute:= FALSE);
				RETURN;
			END_IF
			fbSdoWrite(bExecute:= FALSE);
		END_IF
	ELSE
		IF bNewCamDelay THEN
			bNewCamDelay := FALSE;
			bSendCamDelay := TRUE;
		END_IF
	END_IF

	IF bSendStrobDelay THEN
		IF bSendStrobDelayFlag XOR fbSdoWrite.bBusy THEN
			bSendStrobDelayFlag := FALSE;
			pFbMultiZ^.stStrobTrigger.nStrobDelay := nStrobDelay;
			fbSdoWrite(sADSNetID:= pFbMultiZ^.P_sAdsNetId, nPortNr:= pFbMultiZ^.P_nAdsPort,
						nIndex:= cPiezoStrobDelay.nIndex, nSubIndex:= cPiezoStrobDelay.nSubIndex, 
						nDataLength:= cPiezoStrobDelay.nLength, nData:= pFbMultiZ^.stStrobTrigger.nStrobDelay, bExecute:= TRUE);							
		END_IF
		IF NOT fbSdoWrite.bBusy THEN
			nSendPauseCnt := 0;
			bSendStrobDelayFlag := TRUE;
			bSendStrobDelay := FALSE;
			IF fbSdoWrite.bError THEN
				stError.Cmd := 0;
				stError.ObjectId := nObjectID;
				stError.POU := E_POU.POU_FB_Stroboscope;
				fbSdoWrite(bExecute:= FALSE);
				RETURN;
			END_IF
			fbSdoWrite(bExecute:= FALSE);
		END_IF
	ELSE
		IF bNewStrobDelay THEN
			bNewStrobDelay := FALSE;
			bSendStrobDelay := TRUE;
		END_IF		
	END_IF
	
	IF bSendStrobDelay2 THEN
		IF bSendStrobDelay2Flag XOR fbSdoWrite.bBusy THEN
			bSendStrobDelay2Flag := FALSE;
			pFbMultiZ^.stStrobTrigger.nStrobDelay2 := nStrobDelay2;
			fbSdoWrite(sADSNetID:= pFbMultiZ^.P_sAdsNetId, nPortNr:= pFbMultiZ^.P_nAdsPort,
						nIndex:= cPiezoStrobDelay2.nIndex, nSubIndex:= cPiezoStrobDelay2.nSubIndex, 
						nDataLength:= cPiezoStrobDelay2.nLength, nData:= pFbMultiZ^.stStrobTrigger.nStrobDelay2, bExecute:= TRUE);							
		END_IF
		IF NOT fbSdoWrite.bBusy THEN
			nSendPauseCnt := 0;
			bSendStrobDelay2Flag := TRUE;
			bSendStrobDelay2 := FALSE;
			IF fbSdoWrite.bError THEN
				stError.Cmd := 0;
				stError.ObjectId := nObjectID;
				fbSdoWrite(bExecute:= FALSE);
				RETURN;
			END_IF
			fbSdoWrite(bExecute:= FALSE);
		END_IF
	ELSE
		IF bNewStrobDelay2 THEN
			bNewStrobDelay2 := FALSE;
			bSendStrobDelay2 := TRUE;
		END_IF			
	END_IF
	
	IF bSendDroplist1_4 THEN
		IF bSendDroplist1_4Flag XOR fbSdoWrite.bBusy THEN
			bSendDroplist1_4Flag := FALSE;
			pFbMultiZ^.stStrobTrigger.aDroplist := aDroplist; 
			MEMCPY(ADR(fbSdoWrite.nData),ADR(pFbMultiZ^.stStrobTrigger.aDroplist[1]),4);			
			fbSdoWrite(sADSNetID:= pFbMultiZ^.P_sAdsNetId, nPortNr:= pFbMultiZ^.P_nAdsPort,
						nIndex:= cPiezoStrobDroplist1_4.nIndex, nSubIndex:= cPiezoStrobDroplist1_4.nSubIndex, 
						nDataLength:= cPiezoStrobDroplist1_4.nLength, bExecute:= TRUE);								
		END_IF
		IF NOT fbSdoWrite.bBusy THEN
			nSendPauseCnt := 0;
			bSendDroplist1_4Flag := TRUE;
			bSendDroplist1_4 := FALSE;
			IF fbSdoWrite.bError THEN
				stError.Cmd := 0;
				stError.ObjectId := nObjectID;
				fbSdoWrite(bExecute:= FALSE);
				RETURN;
			END_IF
			fbSdoWrite(bExecute:= FALSE);
		END_IF
		IF bNewDroplist1_4 THEN
			bNewDroplist1_4 := FALSE;
			bSendDroplist1_4 := TRUE;
		END_IF			
	END_IF
	
	IF bSendDroplist5_8 THEN
		IF bSendDroplist5_8Flag XOR fbSdoWrite.bBusy THEN
			bSendDroplist5_8Flag := FALSE;
			pFbMultiZ^.stStrobTrigger.aDroplist := aDroplist; 
			MEMCPY(ADR(fbSdoWrite.nData),ADR(pFbMultiZ^.stStrobTrigger.aDroplist[5]),4);		
			fbSdoWrite(sADSNetID:= pFbMultiZ^.P_sAdsNetId, nPortNr:= pFbMultiZ^.P_nAdsPort,
						nIndex:= cPiezoStrobDroplist5_8.nIndex, nSubIndex:= cPiezoStrobDroplist5_8.nSubIndex, 
						nDataLength:= cPiezoStrobDroplist5_8.nLength, bExecute:= TRUE);								
								
		END_IF
		IF NOT fbSdoWrite.bBusy THEN
			nSendPauseCnt := 0;
			bSendDroplist5_8Flag := TRUE;
			bSendDroplist5_8 := FALSE;
			IF fbSdoWrite.bError THEN
				stError.Cmd := 0;
				stError.ObjectId := nObjectID;
				fbSdoWrite(bExecute:= FALSE);
				RETURN;
			END_IF
			fbSdoWrite(bExecute:= FALSE);
		END_IF
	ELSE
		IF bNewDroplist5_8 THEN
			bNewDroplist5_8 := FALSE;
			bSendDroplist5_8 := TRUE;
		END_IF			
	END_IF
	
	IF bSendDroplist9_12 THEN
		IF bSendDroplist9_12Flag XOR fbSdoWrite.bBusy THEN
			bSendDroplist9_12Flag := FALSE;
			pFbMultiZ^.stStrobTrigger.aDroplist := aDroplist; 
			MEMCPY(ADR(fbSdoWrite.nData),ADR(pFbMultiZ^.stStrobTrigger.aDroplist[9]),4);
			fbSdoWrite(sADSNetID:= pFbMultiZ^.P_sAdsNetId, nPortNr:= pFbMultiZ^.P_nAdsPort,
						nIndex:= cPiezoStrobDroplist9_12.nIndex, nSubIndex:= cPiezoStrobDroplist9_12.nSubIndex, 
						nDataLength:= cPiezoStrobDroplist9_12.nLength, bExecute:= TRUE);								
								
		END_IF
		IF NOT fbSdoWrite.bBusy THEN
			nSendPauseCnt := 0;
			bSendDroplist9_12Flag := TRUE;
			bSendDroplist9_12 := FALSE;
			IF fbSdoWrite.bError THEN
				stError.Cmd := 0;
				stError.ObjectId := nObjectID;
				fbSdoWrite(bExecute:= FALSE);
				RETURN;
			END_IF
			fbSdoWrite(bExecute:= FALSE);
		END_IF
	ELSE
		IF bNewDroplist9_12 THEN
			bNewDroplist9_12 := FALSE;
			bSendDroplist9_12 := TRUE;
		END_IF			
	END_IF
	
	IF bSendDroplist13_16 THEN
		IF bSendDroplist13_16Flag XOR fbSdoWrite.bBusy THEN
			bSendDroplist13_16Flag := FALSE;
			pFbMultiZ^.stStrobTrigger.aDroplist := aDroplist; 
			MEMCPY(ADR(fbSdoWrite.nData),ADR(pFbMultiZ^.stStrobTrigger.aDroplist[13]),4);
			fbSdoWrite(sADSNetID:= pFbMultiZ^.P_sAdsNetId, nPortNr:= pFbMultiZ^.P_nAdsPort,
						nIndex:= cPiezoStrobDroplist13_16.nIndex, nSubIndex:= cPiezoStrobDroplist13_16.nSubIndex, 
						nDataLength:= cPiezoStrobDroplist13_16.nLength, bExecute:= TRUE);
		END_IF
		IF NOT fbSdoWrite.bBusy THEN
			nSendPauseCnt := 0;
			bSendDroplist13_16Flag := TRUE;
			bSendDroplist13_16 := FALSE;
			IF fbSdoWrite.bError THEN
				stError.Cmd := 0;
				stError.ObjectId := nObjectID;
				fbSdoWrite(bExecute:= FALSE);
				RETURN;
			END_IF
			fbSdoWrite(bExecute:= FALSE);
		END_IF
	ELSE
		IF bNewDroplist13_16 THEN
			bNewDroplist13_16 := FALSE;
			bSendDroplist13_16 := TRUE;
		END_IF		
	END_IF
END_IF

//Prozessdaten aktualisieren
stProcessData.nObjId := nObjectID;
stProcessData.n32Data[0] := BOOL_TO_DINT(bIsInit);
stProcessData.n32Data[1] := eCurrentState;
stProcessData.n32Data[2] := stError.ErrorId;

aObjProcData[nNotifyId] := stProcessData;

ACTION A_StrobTest:
CASE nStateA_StrobTest OF
	0:	//Einschalten
		IF bSendStrobTestFlag XOR fbSdoWrite.bBusy THEN
			bSendStrobTestFlag := FALSE;
			pFbMultiZ^.stStrobTrigger.bTest := TRUE;
			//fbMultiZSendSdoVar(pFbMultiZ:= pFbMultiZ, eSdoVariType:= E_MzSdoVariType.VARITYPE_PiezoStrobTest, bExecute:= TRUE);
			fbSdoWrite(sADSNetID:= pFbMultiZ^.P_sAdsNetId, nPortNr:= pFbMultiZ^.P_nAdsPort,
					nIndex:= cPiezoStrobTest.nIndex, nSubIndex:= cPiezoStrobTest.nSubIndex, 
					nDataLength:= cPiezoStrobTest.nLength, nData:= 1, bExecute:= TRUE);
		END_IF

		IF NOT fbSdoWrite.bBusy THEN
			bSendStrobTestFlag := TRUE;
			IF fbSdoWrite.bError THEN
				stError.ErrorId := fbSdoWrite.nAdsErrorId;
				stError.POUState := nStateA_StrobTest;
				nStateA_StrobTest := 99;
			ELSE
				nStateA_StrobTest := 1;	
			END_IF
			fbSdoWrite(bExecute:= FALSE);
		END_IF
		
	1:	//Warten auf Auschaltbefehl
		IF NOT bStrobTestCtrl THEN
			IF bSendStrobTestFlag XOR fbSdoWrite.bBusy THEN
				bSendStrobTestFlag := FALSE;
				pFbMultiZ^.stStrobTrigger.bTest := FALSE;
				//fbMultiZSendSdoVar(pFbMultiZ:= pFbMultiZ, eSdoVariType:= E_MzSdoVariType.VARITYPE_PiezoStrobTest, bExecute:= TRUE);
				fbSdoWrite(sADSNetID:= pFbMultiZ^.P_sAdsNetId, nPortNr:= pFbMultiZ^.P_nAdsPort,
						nIndex:= cPiezoStrobTest.nIndex, nSubIndex:= cPiezoStrobTest.nSubIndex, 
						nDataLength:= cPiezoStrobTest.nLength, nData:= 0, bExecute:= TRUE);
			END_IF
			
			IF NOT fbSdoWrite.bBusy THEN
				bSendStrobTestFlag := TRUE;
				IF fbSdoWrite.bError THEN
					stError.ErrorId := fbSdoWrite.nAdsErrorId;
					stError.POUState := nStateA_StrobTest;
					nStateA_StrobTest := 99;
				ELSE
					nStateA_StrobTest := 80;	
				END_IF
				fbSdoWrite(bExecute:= FALSE);
			END_IF
		END_IF

	70:	//Abbrechen
		IF NOT bSendStrobTestFlag THEN	//letzte SDO-Send ist noch nicht abgearbeitet
			fbSdoWrite(bExecute:= FALSE);
		END_IF
		bSendStrobTestFlag := TRUE;
		nStateA_StrobTest := 71;
		
	71:	//Ausschaltbefehl senden
		IF bSendStrobTestFlag XOR fbSdoWrite.bBusy THEN
			bSendStrobTestFlag := FALSE;
			pFbMultiZ^.stStrobTrigger.bTest := FALSE;
			//fbMultiZSendSdoVar(pFbMultiZ:= pFbMultiZ, eSdoVariType:= E_MzSdoVariType.VARITYPE_PiezoStrobTest, bExecute:= TRUE);
			fbSdoWrite(sADSNetID:= pFbMultiZ^.P_sAdsNetId, nPortNr:= pFbMultiZ^.P_nAdsPort,
					nIndex:= cPiezoStrobTest.nIndex, nSubIndex:= cPiezoStrobTest.nSubIndex, 
					nDataLength:= cPiezoStrobTest.nLength, nData:= 0, bExecute:= TRUE);
			
		END_IF
		IF NOT fbSdoWrite.bBusy THEN
			bSendStrobTestFlag := TRUE;
			IF fbSdoWrite.bError THEN
				stError.ErrorId := fbSdoWrite.nAdsErrorId;
				stError.POUState := nStateA_StrobTest;
				nStateA_StrobTest := 99;
			ELSE
				nStateA_StrobTest := 80;	
			END_IF
			fbSdoWrite(bExecute:= FALSE);
		END_IF	
END_CASE

//Errorhandling
IF nStateA_StrobTest = 99 THEN
	stError.Cmd := E_Action.ACTION_StrobTest;
	stError.POUAction := E_POUACT.POUACT_A_StrobTest;
	fbErrorList.M_Add(stError);
END_IF
END_ACTION

METHOD FB_init : BOOL
VAR_INPUT
	bInitRetains : BOOL; // if TRUE, the retain variables are initialized (warm start / cold start)
	bInCopyCode : BOOL;  // if TRUE, the instance afterwards gets moved into the copy code (online change)
END_VAR
eObjectType := E_ObjectType.OBJECTTYPE_Stroboscope;
eObjectGroup := E_ObjectGroup.OBJECTGROUP_Target OR E_ObjectGroup.OBJECTGROUP_Device;
END_METHOD

METHOD M_CancelAction
VAR_INPUT
	eAction : E_Action;
END_VAR
IF eAction = E_Action.ACTION_StrobTest THEN
	IF bStrobTest AND nStateA_StrobTest < 70 THEN
		nStateA_StrobTest := 70;
	END_IF
END_IF
END_METHOD

METHOD M_CheckAction : ERRORID
VAR_INPUT
	refActionData 	: REFERENCE TO ST_ActionData;
	pCorrelObject	: POINTER TO FB_Object;
END_VAR
IF refActionData.eAction = E_Action.ACTION_TeachTarget THEN
	IF NOT DINT_TO_UINT(refActionData.aParams[1]) = E_TargetRef.TARGETREF_SpecPoint AND refActionData.aParams[2] = 1 THEN
		M_CheckAction := E_ErrorIdCmd.ERRORID_InvalidTargetPointRef;
	END_IF
END_IF
END_METHOD

METHOD M_ExeAction : ERRORID
VAR_INPUT
	refActionData : REFERENCE TO ST_ActionData;	
END_VAR
IF refActionData.eAction = E_Action.ACTION_Init THEN
	bIsInit := TRUE;
	RETURN;
ELSIF 
	refActionData.eAction = E_Action.ACTION_StrobTest THEN
	bStrobTestCtrl := refActionData.aParams[1].0;
	//In Action nur treten, wenn:
	IF NOT bStrobTest AND bStrobTestCtrl THEN
		bStrobTest := TRUE;
		bBusy := TRUE;
		eCurrentState := E_MachineState.MACHINESTATE_Active;
	END_IF
ELSIF
	refActionData.eAction = E_Action.ACTION_Stop THEN
	IF bStrobTest THEN
		nStateA_StrobTest := 70;
	END_IF
END_IF
END_METHOD

METHOD M_GetActionBusy : BOOL
VAR_INPUT
	eAction : E_Action;
END_VAR
IF eAction = E_Action.ACTION_StrobTest THEN
	M_GetActionBusy := bStrobTest;
END_IF
END_METHOD

METHOD M_GetAllProps : ERRORID
VAR_INPUT
	refCmdData : REFERENCE TO  ST_CmdData;
END_VAR

VAR
	pData	: POINTER TO ARRAY[1..16] OF USINT;
END_VAR
SUPER^.M_GetAllProps(refCmdData); 
nCurrentPropIndex := nCurrentPropIndex + 1;
refCmdData.n32Data[nCurrentPropIndex] := nMultiZNr;
nCurrentPropIndex := nCurrentPropIndex + 1;
refCmdData.n32Data[nCurrentPropIndex] := nCamDelay;
nCurrentPropIndex := nCurrentPropIndex + 1;
refCmdData.n32Data[nCurrentPropIndex] := nStrobDelay;
nCurrentPropIndex := nCurrentPropIndex + 1;
refCmdData.n32Data[nCurrentPropIndex] := nStrobDelay2;
//Droplist aus aDroplist nach "refCmdData.n32Data[16]" bis "refCmdData.n32Data[19]" übertragen
nCurrentPropIndex := nCurrentPropIndex + 1;
pData := ADR(refCmdData.n32Data[nCurrentPropIndex]);
pData^ := aDroplist;
nCurrentPropIndex := nCurrentPropIndex + 4;
refCmdData.n32Data[nCurrentPropIndex] := nGCodeTargetNr;
END_METHOD

METHOD M_SetAllProps : ERRORID
VAR_INPUT
	refCmdData : REFERENCE TO  ST_CmdData;
END_VAR

VAR
	pData	: POINTER TO ARRAY[1..16] OF USINT;
END_VAR
M_SetAllProps := SUPER^.M_SetAllProps(refCmdData);

IF M_SetAllProps > 0 THEN
	RETURN;
END_IF

nCurrentPropIndex := nCurrentPropIndex + 1;
nMultiZNr := DINT_TO_USINT(refCmdData.n32Data[nCurrentPropIndex]);

pFbMultiZ := ADR(aFbMultiZRef[nMultiZNr]);
nCurrentPropIndex := nCurrentPropIndex + 1;
nCamDelay := DINT_TO_UINT(refCmdData.n32Data[nCurrentPropIndex]);
bNewCamDelay := TRUE;
nCurrentPropIndex := nCurrentPropIndex + 1;
nStrobDelay := DINT_TO_UINT(refCmdData.n32Data[nCurrentPropIndex]);
bNewStrobDelay := TRUE;
nCurrentPropIndex := nCurrentPropIndex + 1;
nStrobDelay2 := DINT_TO_UINT(refCmdData.n32Data[nCurrentPropIndex]);
bNewStrobDelay2 := TRUE;

//Droplist aus "refCmdData.n32Data[16]" bis "refCmdData.n32Data[19]" nach aDroplist übertragen
nCurrentPropIndex := nCurrentPropIndex + 1;
pData := ADR(refCmdData.n32Data[nCurrentPropIndex]);
aDroplist := pData^;
bNewDroplist1_4 := TRUE;
bNewDroplist5_8  := TRUE;
bNewDroplist9_12 := TRUE;
bNewDroplist13_16  := TRUE; 
nCurrentPropIndex := nCurrentPropIndex + 4;
nGCodeTargetNr := DINT_TO_UINT(refCmdData.n32Data[nCurrentPropIndex]);
nNoOfProps := nCurrentPropIndex + 1;
END_METHOD

METHOD M_SetSingleProp : ERRORID
VAR_INPUT
	refCmdData : REFERENCE TO  ST_CmdData;
END_VAR
VAR
	pSource			: POINTER TO ARRAY[1..4] OF USINT;
	pDestination	: POINTER TO ARRAY[1..4] OF USINT;
END_VAR
IF (nSpecPropIndex + 4) = refCmdData.aHeader[1] THEN
	M_SetSingleProp := E_ErrorIdCmd.ERRORID_InvalidProperty;//MultiZNr Triiger darf nicht verändert werden
ELSIF (nSpecPropIndex + 5) = refCmdData.aHeader[1] THEN
	nCamDelay := DINT_TO_UINT(refCmdData.n32Data[0]);
	bNewCamDelay := TRUE;	
ELSIF (nSpecPropIndex + 6) = refCmdData.aHeader[1] THEN
	nStrobDelay := DINT_TO_UINT(refCmdData.n32Data[0]);
	bNewStrobDelay := TRUE;		
ELSIF (nSpecPropIndex + 7) = refCmdData.aHeader[1] THEN
	nStrobDelay2 := DINT_TO_UINT(refCmdData.n32Data[0]);
	bNewStrobDelay2 := TRUE;	
ELSIF (nSpecPropIndex + 8) = refCmdData.aHeader[1] THEN
	pSource := ADR(refCmdData.n32Data[0]);
	pDestination := ADR(aDroplist[1]);
	pDestination^ := pSource^;	
ELSIF (nSpecPropIndex + 9) = refCmdData.aHeader[1] THEN
	pSource := ADR(refCmdData.n32Data[0]);
	pDestination := ADR(aDroplist[5]);
	pDestination^ := pSource^;	
ELSIF (nSpecPropIndex + 10) = refCmdData.aHeader[1] THEN
	pSource := ADR(refCmdData.n32Data[0]);
	pDestination := ADR(aDroplist[9]);
	pDestination^ := pSource^;
ELSIF (nSpecPropIndex + 11) = refCmdData.aHeader[1] THEN
	pSource := ADR(refCmdData.n32Data[0]);
	pDestination := ADR(aDroplist[13]);
	pDestination^ := pSource^;		
ELSE
	M_SetSingleProp := SUPER^.M_SetSingleProp(refCmdData);
END_IF
END_METHOD

METHOD M_Stop : ERRORID
VAR_INPUT
END_VAR
IF nStateA_StrobTest = 1 THEN
 	nStateA_StrobTest := 70;
END_IF
END_METHOD

PROPERTY P_nGCodeTargetNr : UINT
GET
P_nGCodeTargetNr := nGCodeTargetNr;
END_GET
END_PROPERTY

END_FUNCTION_BLOCK

// ---- Objects/Targets/Active/FB_WorkplateCamera.TcPOU
FUNCTION_BLOCK FB_WorkplateCamera EXTENDS FB_ActiveTarget
VAR_INPUT
END_VAR
VAR
	nNoOfSpecPoints 		: USINT;
	stFocusPoint			: ST_3DPoint;
	
	bTakePicture			: BOOL;
	nStateA_TakePicture		: USINT;
	tDelayTakePicture		: TIME;
	timerTakePicture		: TON;
	nRequestArg1			: DINT;
	nRequestArg2			: DINT;
END_VAR

IF eCurrentState = E_MachineState.MACHINESTATE_Active THEN
	IF bTakePicture THEN
		A_TakePicture();
		IF nStateA_TakePicture = 80 THEN
			nStateA_TakePicture := 0;
			bTakePicture := FALSE;
			eCurrentState := E_MachineState.MACHINESTATE_Idle;
		END_IF
	END_IF	
END_IF

//Prozessdaten aktualisieren
stProcessData.nObjId := nObjectID;
stProcessData.n32Data[0] := BOOL_TO_DINT(bIsInit);
stProcessData.n32Data[1] := eCurrentState;
stProcessData.n32Data[2] := stError.ErrorId;
aObjProcData[nNotifyId] := stProcessData;

ACTION A_TakePicture:
IF nStateA_TakePicture = 0 THEN //Timer starten
	timerTakePicture(IN:= TRUE, PT:= tDelayTakePicture);
	IF timerTakePicture.Q THEN
		timerTakePicture(IN:= FALSE);
		stInterResponse.eInteractMessageType := E_InteractMessageType.INTERACTMES_NONE;
		stInteractRequest.eInteractMessageType := E_InteractMessageType.INTERACTMES_WaitForUser;
		stInteractRequest.nObjectId := nObjectID;
		stInteractRequest.nArg1 := nRequestArg1;
		stInteractRequest.nArg2 := nRequestArg2;
		nStateA_TakePicture := 1;
	END_IF
ELSIF nStateA_TakePicture = 1 THEN //Auf InteractResponse warten
	IF stInterResponse.eInteractMessageType = E_InteractMessageType.INTERACTMES_Continue OR 
							stInterResponse.eInteractMessageType = E_InteractMessageType.INTERACTMES_Cancel THEN
		stInteractRequest.eInteractMessageType := E_InteractMessageType.INTERACTMES_NONE;
		nStateA_TakePicture := 80;
	END_IF
ELSIF nStateA_TakePicture = 70 THEN //Abbrechen
	timerTakePicture(IN:= FALSE);
	stInteractRequest.eInteractMessageType := E_InteractMessageType.INTERACTMES_NONE;
	nStateA_TakePicture := 80;
END_IF
END_ACTION

METHOD FB_init : BOOL
VAR_INPUT
	bInitRetains : BOOL; // if TRUE, the retain variables are initialized (warm start / cold start)
	bInCopyCode : BOOL;  // if TRUE, the instance afterwards gets moved into the copy code (online change)
END_VAR
eObjectType := E_ObjectType.OBJECTTYPE_WorkplateCamera;
eObjectGroup := E_ObjectGroup.OBJECTGROUP_Target OR E_ObjectGroup.OBJECTGROUP_Device;
END_METHOD

METHOD M_ApplyPos : ERRORID
VAR_INPUT
	eTargetRef 		: E_TargetRef;
	nPointSlotNr	: UINT;
	stPos 			: ST_3DPoint;
	bXPos			: BOOL;
	bYPos			: BOOL;
	bZPos			: BOOL;	
END_VAR

VAR
	stAbsPos		: ST_3DPoint;
END_VAR
IF eTargetRef = E_TargetRef.TARGETREF_SpecPoint THEN
	IF nPointSlotNr = 1 THEN
		stAbsPos := P_stAbsPosLB;
		IF bXPos THEN
			stFocusPoint.X := stPos.X - stAbsPos.X;	
		END_IF
		IF bYPos THEN
			stFocusPoint.Y := stPos.Y - stAbsPos.Y;	
		END_IF
		IF bZPos THEN
			stFocusPoint.Z := stPos.Z - stAbsPos.Z;	
		END_IF
	ELSE
		M_ApplyPos := E_ErrorIdCmd.ERRORID_InvalidTargetPointNr;
	END_IF
ELSE
	M_ApplyPos := SUPER^.M_ApplyPos(eTargetRef, nPointSlotNr, stPos, bXPos, bYPos, bZPos);
END_IF
END_METHOD

METHOD M_CancelAction
VAR_INPUT
	eAction : E_Action;
END_VAR
END_METHOD

METHOD M_CheckAction : ERRORID
VAR_INPUT
	refActionData 	: REFERENCE TO ST_ActionData;
	pCorrelObject	: POINTER TO FB_Object;
END_VAR
IF refActionData.eAction = E_Action.ACTION_TeachTarget THEN
	IF NOT DINT_TO_UINT(refActionData.aParams[1]) = E_TargetRef.TARGETREF_SpecPoint AND refActionData.aParams[2] = 1 THEN
		M_CheckAction := E_ErrorIdCmd.ERRORID_InvalidTargetPointRef;
	END_IF
END_IF
END_METHOD

METHOD M_CheckProcDataType : BOOL
VAR_INPUT
	eProcDataType : E_ProcDataType;
END_VAR
END_METHOD

METHOD M_ExeAction : ERRORID
VAR_INPUT
	refActionData : REFERENCE TO ST_ActionData;	
END_VAR
IF refActionData.eAction = E_Action.ACTION_Init THEN
	bIsInit := TRUE;
ELSIF refActionData.eAction = E_Action.ACTION_TakePicture THEN
	IF NOT bTakePicture THEN
		tDelayTakePicture := DINT_TO_TIME(refActionData.aParams[1]);
		nRequestArg1 := refActionData.aParams[2];
		nRequestArg2 := refActionData.aParams[3];
		bTakePicture := TRUE;
		eCurrentState := E_MachineState.MACHINESTATE_Active;
		bBusy := TRUE;
	END_IF
ELSE
	M_ExeAction := E_ErrorIdCmd.ERRORID_InvalidAction;
END_IF
END_METHOD

METHOD M_GetAbsPos : ST_3DPoint
VAR_INPUT
	pChildPos	: POINTER TO ST_3DPoint;
	eTargetRef 	: E_TargetRef;
	nParam1		: UINT;
 	nParam2		: UINT;
	nParam3		: USINT;
	nParam4		: USINT;
	nZLevel		: USINT;
END_VAR
VAR_OUTPUT
	nErrorId 	: ERRORID;
	lrAngle		: LREAL;
END_VAR
VAR
	stLocPosLB : ST_3DPoint;
END_VAR
IF eTargetRef = E_TargetRef.TARGETREF_SpecPoint THEN
	IF nParam1 = 1 THEN	//FocusPoint
		stLocPosLB := P_stRelPosLB;
		stLocPosLB := F_Add3DPoints(stLocPosLB,stFocusPoint);
		M_GetAbsPos := pParentTarget^.M_GetAbsPos(pChildPos := ADR(stLocPosLB), eTargetRef:= E_TargetRef.TARGETREF_LeftBottom,
													nParam1:= 0,
													nParam2:= 0, nParam3:= 0, nParam4:= 0, nZLevel:= 0,
													lrAngle => lrAngle, nErrorId=> nErrorId);		
	ELSE
		nErrorId := E_ErrorIdCmd.ERRORID_InvalidTargetPointNr;
	END_IF
ELSE
	M_GetAbsPos := SUPER^.M_GetAbsPos(pChildPos := pChildPos, eTargetRef:= eTargetRef,
													nParam1:= nParam1,
													nParam2:= nParam2, nParam3:= nParam3, nParam4:= 0, nZLevel:= nZLevel,
													lrAngle => lrAngle, nErrorId=> nErrorId);	
END_IF
END_METHOD

METHOD M_GetActionBusy : BOOL
VAR_INPUT
	eAction : E_Action;
END_VAR
IF eAction = E_Action.ACTION_TakePicture AND bTakePicture THEN
	M_GetActionBusy := TRUE;
END_IF
END_METHOD

METHOD M_GetAllProps : ERRORID
VAR_INPUT
	refCmdData : REFERENCE TO  ST_CmdData;
END_VAR

VAR
END_VAR
SUPER^.M_GetAllProps(refCmdData); 

nCurrentPropIndex := nCurrentPropIndex + 1;
refCmdData.n32Data[nCurrentPropIndex] := nNoOfSpecPoints;
nCurrentPropIndex := nCurrentPropIndex + 1;
refCmdData.n32Data[nCurrentPropIndex] := REAL_TO_DINT(stFocusPoint.X);
nCurrentPropIndex := nCurrentPropIndex + 1;
refCmdData.n32Data[nCurrentPropIndex] := REAL_TO_DINT(stFocusPoint.Y);
nCurrentPropIndex := nCurrentPropIndex + 1;
refCmdData.n32Data[nCurrentPropIndex] := REAL_TO_DINT(stFocusPoint.Z);
END_METHOD

METHOD M_GetProcData : DINT
VAR_INPUT
	eProcDataType : E_ProcDataType;
END_VAR
END_METHOD

METHOD M_Reset
END_METHOD

METHOD M_SetAllProps : ERRORID
VAR_INPUT
	refCmdData : REFERENCE TO  ST_CmdData;
END_VAR

VAR
	pData	: POINTER TO ARRAY[1..16] OF USINT;
END_VAR
M_SetAllProps := SUPER^.M_SetAllProps(refCmdData);

IF M_SetAllProps > 0 THEN
	RETURN;
END_IF

nCurrentPropIndex := nCurrentPropIndex + 1;
nSpecPropIndex := nCurrentPropIndex;
nNoOfSpecPoints := DINT_TO_USINT(refCmdData.n32Data[nCurrentPropIndex]);
nCurrentPropIndex := nCurrentPropIndex + 1;
stFocusPoint.X := DINT_TO_REAL(refCmdData.n32Data[nCurrentPropIndex]);
nCurrentPropIndex := nCurrentPropIndex + 1; 
stFocusPoint.Y := DINT_TO_REAL(refCmdData.n32Data[nCurrentPropIndex]);
nCurrentPropIndex := nCurrentPropIndex + 1;
stFocusPoint.Z := DINT_TO_REAL(refCmdData.n32Data[nCurrentPropIndex]);
nNoOfProps := nCurrentPropIndex + 1;
END_METHOD

METHOD M_SetSingleProp : ERRORID
VAR_INPUT
	refCmdData : REFERENCE TO  ST_CmdData;
END_VAR
VAR
	pSource			: POINTER TO ARRAY[1..4] OF USINT;
	pDestination	: POINTER TO ARRAY[1..4] OF USINT;
END_VAR
IF nSpecPropIndex = refCmdData.aHeader[1] THEN
	M_SetSingleProp := E_ErrorIdCmd.ERRORID_InvalidProperty;//Anzahl SpecPoints darf nicht verändert werden
ELSIF (nSpecPropIndex + 1) = refCmdData.aHeader[1] THEN
	stFocusPoint.X := DINT_TO_REAL(refCmdData.n32Data[0]);	
ELSIF (nSpecPropIndex + 2) = refCmdData.aHeader[1] THEN
	stFocusPoint.Y := DINT_TO_REAL(refCmdData.n32Data[0]);
ELSIF (nSpecPropIndex + 3) = refCmdData.aHeader[1] THEN
	stFocusPoint.Z := DINT_TO_REAL(refCmdData.n32Data[0]);
ELSE
	M_SetSingleProp := SUPER^.M_SetSingleProp(refCmdData);
END_IF
END_METHOD

METHOD M_Stop : ERRORID
VAR_INPUT
END_VAR
END_METHOD

END_FUNCTION_BLOCK

// ---- Objects/Targets/Active/FB_MtpHolder.TcPOU
FUNCTION_BLOCK FB_MtpHolder EXTENDS FB_ActiveTarget IMPLEMENTS I_SlotTarget

VAR
	fbSlotList			: FB_SlotList;
	pSlot				: POINTER TO FB_Slot;
	nNumberOfSlots		: UINT;
	nFirstSlotPropIndex	: UINT;	//erster Index für Slots (benötigt in M_SetSingleProps)
	nLastSlotPropIndex	: UINT;	//letzte Index für Slots (benötigt in M_SetSingleProps)

	//Hardware-Verküpfung
	pHeaterRef			: POINTER TO FB_HwRef4ChHeater;
	
	//Prozessdaten
	nTempActual			: UINT;

	//Spec-Properties
	nHeaterChannel		: USINT;
	
	//****************************************Aktionvariablen****************************************************
	
	//Action: "Heating"
	nTempSetpoint		: USINT;	//Bei Mtp-Holder bzw. SubstHolder in ganzen °C
	bHeaterOn			: BOOL;
	
	//Action: "EdgeLight"
	bEdgeLigthOn		: BOOL;
	
END_VAR

IF pHeaterRef = 0 THEN
	RETURN;
END_IF
IF bInitFB THEN
	bInitFB := FALSE;
	stError.ObjectId := nObjectID;
	stError.HardwareGrp := E_HardwareGrp.Nothing;
	stError.POU := E_POU.POU_FB_MtpHolder;
END_IF

CASE eCurrentState OF
	E_MachineState.MACHINESTATE_Active:
		CASE eCurrentAction OF
			E_Action.ACTION_Heating:
				pHeaterRef^.P_nTempSetpoint := nTempSetpoint;
				pHeaterRef^.P_bHeatingOn := bHeaterOn;
				//Hier muss noch eine Abfrage erfolgen, ob Heizer ON
				//dazu braucht es ein PDO vom Heizer
				bBusy := FALSE;
				eCurrentAction := E_Action.ACTION_Nothing;
				eCurrentState:= E_MachineState.MACHINESTATE_Idle;			
			E_Action.ACTION_SwitchLight:
				pHeaterRef^.P_bEdgeLightOn := bEdgeLigthOn;
				//Hier muss noch eine Abfrage erfolgen, ob Heizer ON
				//dazu braucht es ein PDO vom Heizer
				bBusy := FALSE;
				eCurrentAction := E_Action.ACTION_Nothing;
				eCurrentState:= E_MachineState.MACHINESTATE_Idle;			
		END_CASE
END_CASE

//Prozessdaten aktualisieren
stProcessData.nObjId := nObjectID;
stProcessData.n32Data[0] := BOOL_TO_DINT(bIsInit);
stProcessData.n32Data[1] := eCurrentState;
stProcessData.n32Data[2] := stError.ErrorId;
nTempActual := pHeaterRef^.P_nTempActual;
stProcessData.n32Data[3] := BOOL_TO_DINT(pHeaterRef^.P_bHeatingOn);
stProcessData.n32Data[4] := nTempActual;
aObjProcData[nNotifyId] := stProcessData;

METHOD FB_init : BOOL
VAR_INPUT
	bInitRetains : BOOL; // if TRUE, the retain variables are initialized (warm start / cold start)
	bInCopyCode : BOOL;  // if TRUE, the instance afterwards gets moved into the copy code (online change)
END_VAR
eObjectType := E_ObjectType.OBJECTTYPE_MtpHolder;
eObjectGroup := E_ObjectGroup.OBJECTGROUP_Target OR E_ObjectGroup.OBJECTGROUP_Device;
END_METHOD

METHOD M_AddChild : ERRORID
VAR_INPUT
	pObject : POINTER TO FB_Object;
	nSlotNr	: UINT;
	nIndex 	: INT;	
END_VAR

VAR
	pSlot : POINTER TO FB_Slot;
END_VAR
//In den abgeleiteten Tool-FBs wird überprüft, ob das entsprechende Objekt als Child tauglich ist
IF pObject > 0 THEN
	IF nSlotNr > 0 THEN
		pSlot := fbSlotList.M_GetAtNr(nSlotNr);
		IF pSlot > 0 THEN
			IF pSlot^.P_pChild = 0 THEN
				//Object darf selber noch an keinem Parent hängen
				IF pObject^.P_pParentObject = 0 THEN
					pSlot^.P_pChild := pObject;
					pObject^.P_pObjCollectNode := pObjCollectNode^.nodes.M_AddNewNode(pObject,nIndex);
					pObject^.M_UpdateParent();
				ELSE
					M_AddChild := E_ErrorIdObjMgmt.ERRORID_ObjectAlreadyOnAnotherParent;
				END_IF
			ELSE //Slot bereits belegt
				M_AddChild := E_ErrorIdObjMgmt.ERRORID_SlotIsAlreadyOccupied;
			END_IF		
		ELSE
			M_AddChild := E_ErrorIdObjMgmt.ERRORID_InvalidSlotNumber;			
		END_IF	
	ELSE
		M_AddChild := SUPER^.M_AddChild(pObject,nSlotNr,nIndex);
	END_IF
ELSE
	M_AddChild := E_ErrorIdObjMgmt.ERRORID_InvalidParentObject;
END_IF
END_METHOD

METHOD M_CheckAction : ERRORID
VAR_INPUT
	refActionData 	: REFERENCE TO ST_ActionData;
	pCorrelObject	: POINTER TO FB_Object;
END_VAR
IF NOT refActionData.eAction = E_Action.ACTION_MoveToTarget THEN
	M_CheckAction := E_ErrorIdCmd.ERRORID_InvalidAction;	
END_IF
END_METHOD

METHOD M_CheckProcDataType : BOOL
VAR_INPUT
	eProcDataType : E_ProcDataType;
END_VAR
IF eProcDataType = E_ProcDataType.PROCDATATYPE_Temp1 THEN
	M_CheckProcDataType := TRUE;
END_IF
END_METHOD

METHOD M_ClearAllProps
VAR_INPUT
	bIgnoreParent : BOOL; //Es wird das gesamte OD gelöscht. -> Zeiger auf Parent nicht mehr gültig!
END_VAR
fbSlotList.M_Reset();
SUPER^.M_ClearAllProps(bIgnoreParent);
END_METHOD

METHOD M_ExeAction : ERRORID
VAR_INPUT
	refActionData	: REFERENCE TO ST_ActionData;	
END_VAR
IF pHeaterRef = 0 THEN
	//M_ExeAction := E_ErrorIdObjMgmt.ERRORID_IsNoDevice;
	RETURN;
END_IF
CASE refActionData.eAction OF
	E_Action.ACTION_Init:
		IF pHeaterRef^.P_bNodeEnabled = 0 THEN
			bIsInit := FALSE;
			stError.Cmd := E_Action.ACTION_Init;
			stError.ErrorId := E_ErrorIdCan.ERRORID_NodeNotFound;
			stError.ObjectId := nObjectID;
			fbErrorList.M_Add(stError);
		ELSE
			bIsInit := TRUE;
		END_IF

	E_Action.ACTION_Heating:	//Heizung ON/OFF
		nTempSetpoint := DINT_TO_USINT(refActionData.aParams[1]/10);
		bHeaterOn := DINT_TO_BOOL(refActionData.aParams[2]);
		IF nTempSetpoint > 170 THEN
			M_ExeAction := E_ErrorIdCmd.ERRORID_InvalidHeatingTemp;
		END_IF		
		eCurrentAction := E_Action.ACTION_Heating;
		eCurrentState:= E_MachineState.MACHINESTATE_Active;
		bBusy := TRUE;
		
	E_Action.ACTION_SwitchLight:	//Seitenlicht ON/OFF
		bEdgeligthOn := DINT_TO_BOOL(refActionData.aParams[1]);
		eCurrentAction := E_Action.ACTION_SwitchLight;
		eCurrentState:= E_MachineState.MACHINESTATE_Active;
		bBusy := TRUE;
	ELSE
		M_ExeAction := E_ErrorIdCmd.ERRORID_InvalidAction;	
END_CASE
END_METHOD

METHOD M_GetAbsPos : ST_3DPoint
VAR_INPUT
	pChildPos	: POINTER TO ST_3DPoint;
	eTargetRef 	: E_TargetRef;
	nParam1		: UINT;
 	nParam2		: UINT;
	nParam3		: USINT;
	nParam4		: USINT;
	nZLevel		: USINT;
END_VAR
VAR_OUTPUT
	nErrorId 	: ERRORID;
	lrAngle		: LREAL;
END_VAR
VAR
	stLocPos : ST_3DPoint;
	pSlot : POINTER TO FB_Slot;
END_VAR
IF eTargetRef = E_TargetRef.TARGETREF_Slot THEN
	//Slotnummer checken
	pSlot := M_GetSlot(nParam1);
	IF pSlot > 0 THEN
		stLocPos := F_Add3DPoints(pSlot^.P_stRelPos,stRelPos);
		stLocPos.Z := stLocPos.Z + stDimension.Height;
		//kann es mal sein, dass hier das ParentTarget = 0 ist?
		//ja -> bei der Workplate
		IF pChildPos > 0 THEN
			stLocPos := F_Add3DPoints(stLocPos,pChildPos^);
		END_IF
		IF pParentTarget > 0 THEN
			IF pParentSlot > 0 THEN
				M_GetAbsPos := pParentTarget^.M_GetAbsPos(pChildPos := ADR(stLocPos), eTargetRef:= E_TargetRef.TARGETREF_Slot,
															nParam1:= pParentSlot^.P_nNr,
															nParam2:= 0, nParam3:= 0, nParam4:= 0, nZLevel:= 0, lrAngle=> lrAngle,
															nErrorId=> nErrorId);		
			ELSE
				M_GetAbsPos := pParentTarget^.M_GetAbsPos(pChildPos := ADR(stLocPos), eTargetRef:= E_TargetRef.TARGETREF_LeftBottom,
																nParam1:= 0,
																nParam2:= 0, nParam3:= 0,nParam4:= 0, nZLevel:= 0,
																lrAngle => lrAngle, nErrorId=> nErrorId);
			END_IF
		ELSE
			M_GetAbsPos := stLocPos;
		END_IF		
	ELSE
		nErrorId := E_ErrorIdCmd.ERRORID_InvalidTargetSlot;
	END_IF
	
ELSE
	M_GetAbsPos := SUPER^.M_GetAbsPos(pChildPos := pChildPos, eTargetRef:= eTargetRef,
													nParam1:= nParam1,
													nParam2:= nParam2, nParam3:= nParam3, nParam4:= 0, nZLevel:= nZLevel,
													lrAngle => lrAngle, nErrorId=> nErrorId);	
END_IF
END_METHOD

METHOD M_GetActionBusy : BOOL
VAR_INPUT
	eAction : E_Action;
END_VAR
IF eAction = eCurrentAction THEN
	M_GetActionBusy := TRUE;
END_IF
END_METHOD

METHOD M_GetAllProps : ERRORID
VAR_INPUT
	refCmdData : REFERENCE TO  ST_CmdData;
END_VAR

VAR
	i : UINT;
	pSlot		: POINTER TO FB_Slot;
END_VAR
SUPER^.M_GetAllProps(refCmdData);

nCurrentPropIndex := nCurrentPropIndex + 1;

refCmdData.n32Data[nCurrentPropIndex] := fbSlotList.P_nCount;

fbSlotList.M_SetCurrentToHead();

FOR i := 1 TO fbSlotList.P_nCount BY 1 DO
	pSlot := fbSlotList.M_GetNext();
	IF pSlot > 0 THEN
		nCurrentPropIndex := nCurrentPropIndex + 1;
		refCmdData.n32Data[nCurrentPropIndex] := pSlot^.P_nNr;
		nCurrentPropIndex := nCurrentPropIndex + 1;
		refCmdData.n32Data[nCurrentPropIndex] := REAL_TO_DINT(pSlot^.P_rRelPosX);
		nCurrentPropIndex := nCurrentPropIndex + 1;
		refCmdData.n32Data[nCurrentPropIndex] := REAL_TO_DINT(pSlot^.P_rRelPosY);
		nCurrentPropIndex := nCurrentPropIndex + 1;
		refCmdData.n32Data[nCurrentPropIndex] := REAL_TO_DINT(pSlot^.P_rRelPosZ);
	END_IF		
END_FOR	

nCurrentPropIndex := nCurrentPropIndex + 1;
refCmdData.n32Data[nCurrentPropIndex] := nHeaterChannel;
IF pHeaterRef > 0 THEN
	nCurrentPropIndex := nCurrentPropIndex + 1;
	refCmdData.n32Data[nCurrentPropIndex] := pHeaterRef^.P_nPidKp;
	nCurrentPropIndex := nCurrentPropIndex + 1;
	refCmdData.n32Data[nCurrentPropIndex] := pHeaterRef^.P_nPidKi;
	nCurrentPropIndex := nCurrentPropIndex + 1;
	refCmdData.n32Data[nCurrentPropIndex] := pHeaterRef^.P_nPidKd;
	nCurrentPropIndex := nCurrentPropIndex + 1;
	refCmdData.n32Data[nCurrentPropIndex] := pHeaterRef^.P_nPidTa;
ELSE
	nCurrentPropIndex := nCurrentPropIndex + 1;
	refCmdData.n32Data[nCurrentPropIndex] := 0;
	nCurrentPropIndex := nCurrentPropIndex + 1;
	refCmdData.n32Data[nCurrentPropIndex] := 0;
	nCurrentPropIndex := nCurrentPropIndex + 1;
	refCmdData.n32Data[nCurrentPropIndex] := 0;
	nCurrentPropIndex := nCurrentPropIndex + 1;
	refCmdData.n32Data[nCurrentPropIndex] := 0;
END_IF
END_METHOD

METHOD M_GetProcData : DINT
VAR_INPUT
	eProcDataType : E_ProcDataType;
END_VAR
IF eProcDataType = E_ProcDataType.PROCDATATYPE_Temp1 THEN
	M_GetProcData := nTempActual;
END_IF
END_METHOD

METHOD M_GetSlot : POINTER TO FB_Slot
VAR_INPUT
	nSlotNr : UINT;
END_VAR
M_GetSlot := fbSlotList.M_GetAtNr(nSlotNr);
END_METHOD

METHOD M_GetSlotFromChild : POINTER TO FB_Slot
VAR_INPUT
	pObject : POINTER TO FB_Object;
END_VAR

VAR
	pSlot : POINTER TO FB_Slot;
END_VAR
//Die SlotList iterieren und vergleichen ob Objekte übereinstimmen
fbSlotList.M_SetCurrentToHead();
REPEAT
	pSlot := fbSlotList.M_GetNext();
	IF pSlot > 0 THEN
		IF pSlot^.P_pChild = pObject THEN
			M_GetSlotFromChild := pSlot;
			EXIT;
		END_IF
	END_IF
UNTIL pSlot = 0
END_REPEAT
END_METHOD

METHOD M_SetAllProps : ERRORID
VAR_INPUT
	refCmdData : REFERENCE TO  ST_CmdData;
END_VAR

VAR
	i : UINT;
	pSlot 		: POINTER TO FB_Slot;
END_VAR
M_SetAllProps := SUPER^.M_SetAllProps(refCmdData);

IF M_SetAllProps > 0 THEN
	RETURN;
END_IF

//Slots parametrieren
nCurrentPropIndex := nCurrentPropIndex + 1;
nFirstSlotPropIndex := nCurrentPropIndex;
nNumberOfSlots := DINT_TO_UINT(refCmdData.n32Data[nCurrentPropIndex]);

//Falls SlotList noch nicht existiert, dann neue erstellen
IF fbSlotList.P_nCount = 0 THEN
	FOR i:= 1 TO nNumberOfSlots BY 1 DO
		pSlot := __NEW(FB_Slot(pOwner := THIS));
		fbSlotList.M_Add(pSlot);
		nCurrentPropIndex := nCurrentPropIndex + 1;
		pSlot^.P_nNr := DINT_TO_USINT(refCmdData.n32Data[nCurrentPropIndex]);
		nCurrentPropIndex := nCurrentPropIndex + 1;
		pSlot^.P_rRelPosX := DINT_TO_REAL(refCmdData.n32Data[nCurrentPropIndex]);
		nCurrentPropIndex := nCurrentPropIndex + 1;
		pSlot^.P_rRelPosY := DINT_TO_REAL(refCmdData.n32Data[nCurrentPropIndex]);
		nCurrentPropIndex := nCurrentPropIndex + 1;
		pSlot^.P_rRelPosZ := DINT_TO_REAL(refCmdData.n32Data[nCurrentPropIndex]);
	END_FOR
ELSE
	IF nNumberOfSlots <> fbSlotList.P_nCount THEN	//Anzahl der Slots dürfen sich nicht ändern
		M_SetAllProps := E_ErrorIdObjMgmt.ERRORID_ChangeNoOfSlotsNotAllowed;
		RETURN;		
	END_IF

	FOR i:= 1 TO nNumberOfSlots BY 1 DO
		nCurrentPropIndex := nCurrentPropIndex + 1;
		pSlot := fbSlotList.M_GetAtNr(DINT_TO_USINT(refCmdData.n32Data[nCurrentPropIndex]));
		IF pSlot > 0 THEN
			nCurrentPropIndex := nCurrentPropIndex + 1;
			pSlot^.P_rRelPosX := DINT_TO_REAL(refCmdData.n32Data[nCurrentPropIndex]);
			nCurrentPropIndex := nCurrentPropIndex + 1;
			pSlot^.P_rRelPosY := DINT_TO_REAL(refCmdData.n32Data[nCurrentPropIndex]);
			nCurrentPropIndex := nCurrentPropIndex + 1;
			pSlot^.P_rRelPosZ := DINT_TO_REAL(refCmdData.n32Data[nCurrentPropIndex]);
		ELSE
			M_SetAllProps := 222;
			RETURN;
		END_IF	
	END_FOR
END_IF
nLastSlotPropIndex := nCurrentPropIndex;
nNoOfProps := nCurrentPropIndex + 1;

nCurrentPropIndex := nCurrentPropIndex + 1;
nSpecPropIndex := nCurrentPropIndex;
{IF defined (variable:afbMtpHeatRef)}
IF refCmdData.n32Data[nCurrentPropIndex] > 0 AND refCmdData.n32Data[nCurrentPropIndex] <= cNoOfMtpHeaters THEN
		nHeaterChannel := DINT_TO_USINT(refCmdData.n32Data[nCurrentPropIndex]);
		pHeaterRef := ADR(afbMtpHeatRef[nHeaterChannel]);
		nCurrentPropIndex := nCurrentPropIndex + 1;
		pHeaterRef^.P_nPidKp := DINT_TO_UINT(refCmdData.n32Data[nCurrentPropIndex]);
		nCurrentPropIndex := nCurrentPropIndex + 1;
		pHeaterRef^.P_nPidKi := DINT_TO_UINT(refCmdData.n32Data[nCurrentPropIndex]);
		nCurrentPropIndex := nCurrentPropIndex + 1;
		pHeaterRef^.P_nPidKd := DINT_TO_UINT(refCmdData.n32Data[nCurrentPropIndex]);
		nCurrentPropIndex := nCurrentPropIndex + 1;
		pHeaterRef^.P_nPidTa := DINT_TO_USINT(refCmdData.n32Data[nCurrentPropIndex]);
ELSIF refCmdData.n32Data[nCurrentPropIndex] = 0 THEN
	nCurrentPropIndex := nCurrentPropIndex + 4;
	nHeaterChannel := 0;
	pHeaterRef := 0;
ELSE
	M_SetAllProps := E_ErrorIdObjMgmt.ERRORID_InvalidHeaterChannel;
END_IF
{ELSE}
IF refCmdData.n32Data[nCurrentPropIndex] > 0 THEN
	M_SetAllProps := E_ErrorIdObjMgmt.ERRORID_InvalidHardwareRef;
	RETURN;
END_IF
{END_IF}
nNoOfProps := nCurrentPropIndex + 1;
END_METHOD

METHOD M_Stop : ERRORID
VAR_INPUT
END_VAR
END_METHOD

PROPERTY P_bStopAllOnError : BOOL
GET
END_GET
END_PROPERTY

PROPERTY P_eCurrentState : E_MachineState
GET
END_GET
SET
END_SET
END_PROPERTY

END_FUNCTION_BLOCK

// ---- Hardware/4ChannelHeater/FB_HwRef4ChHeater.TcPOU
FUNCTION_BLOCK FB_HwRef4ChHeater EXTENDS FB_CanNodeBase
VAR_INPUT
END_VAR
VAR_OUTPUT
END_VAR
VAR
	//Eingänge
	nTempActual 	AT %I* : UINT;	//aktuelle Temperatur in 1/100tel °C 
	bTempCutoff 	AT %I* : BOOL;	//Übertemperaturabschaltung wurde aktiviert
	//Ausgänge
	nPidKp 			AT %Q* : UINT; 	//PID-Reglerparameter KP
	nPidKi 			AT %Q* : UINT;	//PID-Reglerparameter KI
	nPidKd 			AT %Q* : UINT;	//PID-Reglerparameter KD
	nPidTa 			AT %Q* : USINT;	//PID-Reglerparameter TA
	bHeatingOn		AT %Q* : BOOL;	//Heizer EIN
	nTempSetpoint	AT %Q* : USINT;	//Solltemperatur in °C (ohne Kommastellen)
	bEdgeLightOn	AT %Q* : BOOL;	//Seitenlicht für Kamera EIN (nur bei Mtp)
END_VAR

IF bNodeEnabled THEN
	SUPER^();
END_IF

PROPERTY P_nPidKp : UINT
SET
nPidKp := P_nPidKp;
END_SET
GET
P_nPidKp := nPidKp;
END_GET
END_PROPERTY

PROPERTY P_nPidKd : UINT
SET
nPidKd := P_nPidKd;
END_SET
GET
P_nPidKd := nPidKd;
END_GET
END_PROPERTY

PROPERTY P_bHeatingOn : BOOL
GET
P_bHeatingOn := bHeatingOn;
END_GET
SET
bHeatingOn := P_bHeatingOn;
END_SET
END_PROPERTY

PROPERTY P_nTempSetpoint : USINT
GET
P_nTempSetpoint := nTempSetpoint;
END_GET
SET
nTempSetpoint := P_nTempSetpoint;
END_SET
END_PROPERTY

PROPERTY P_nPidKi : UINT
GET
P_nPidKi := nPidKi;
END_GET
SET
nPidKi := P_nPidKi;
END_SET
END_PROPERTY

ACTION A_ResetApp:
IF nStateA_ResetApp = 0 THEN
	fbSdoWrite(sADSNetID:= stAdsAdress.sNetId, nPortNr:= stAdsAdress.nPort,
				nIndex := cUpdateRequest.nIndex, nSubIndex := 0, nDataLength := 1, nData:= 1, bExecute:= TRUE);
	IF NOT fbSdoWrite.bBusy THEN
		IF fbSdoWrite.bError THEN
			nErrorId := fbSdoWrite.nAdsErrorId;
			nErrorId2 := fbSdoWrite.nSdoErrorId;
			nStateA_ResetApp := 99;  //Error
		ELSE
			nStateA_ResetApp := 80;
		END_IF
		fbSdoWrite(bExecute:= FALSE);
	END_IF
END_IF
END_ACTION

PROPERTY P_bTempCutoff : BOOL
GET
P_bTempCutoff := bTempCutoff;
END_GET
END_PROPERTY

PROPERTY P_bEdgeLightOn : BOOL
SET
bEdgeLightOn := P_bEdgeLightOn;
END_SET
GET
P_bEdgeLightOn := bEdgeLightOn;
END_GET
END_PROPERTY

PROPERTY P_nTempActual : UINT
GET
P_nTempActual := nTempActual;
END_GET
END_PROPERTY

PROPERTY P_nPidTa : USINT
GET
P_nPidTa := nPidTa;
END_GET
SET
nPidTa := P_nPidTa;
END_SET
END_PROPERTY

END_FUNCTION_BLOCK

// ---- Objects/Targets/Active/FB_SubstHolder.TcPOU
FUNCTION_BLOCK FB_SubstHolder EXTENDS FB_ActiveTarget IMPLEMENTS I_SlotTarget

VAR
	fbSlotList			: FB_SlotList;
	nNumberOfSlots		: UINT;
	nFirstSlotPropIndex	: UINT;	//erster Index für Slots (benötigt in M_SetSingleProps)
	nLastSlotPropIndex	: UINT;	//letzte Index für Slots (benötigt in M_SetSingleProps)

	//Hardware-Verküpfung
	pHeaterRef			: POINTER TO FB_HwRef4ChHeater;

	//Prozessdaten
	bVacuumOk			: BOOL;
	nTempActual			: UINT;

	//Spec-Properties
	nHeaterChannel		: USINT;
	nValveNrCool		: USINT;	//VentilNr Kühlung (FBox)
	nValveNrVac			: USINT;	//VentilNr Vakuum (FBox)
	
	//****************************************Aktionvariablen****************************************************
	
	//Action: "Heating"
	bHeating			: BOOL;		//Action A_Heating() aktiv setzen
	nStateA_Heating		: USINT;	//State von A_Heating()
	nTempHeating		: USINT;	//Bei Mtp-Holder bzw. SubstHolder in ganzen °C
	bHeaterOn			: BOOL;
	

	//Action: "Cooling"
	bCooling			: BOOL;		//Action A_Cooling() aktiv setzen
	nStateA_Cooling		: USINT;	//State von A_Cooling()
	nTempCooling		: UINT;		//Bei Mtp-Holder bzw. SubstHolder in 10tel °C
	bCoolingOn			: BOOL;
	timerCooling		: TON;
	
	//Action: "EdgeLight"
	bEdgeLigthOn		: BOOL;
	
END_VAR

IF bInitFB THEN
	bInitFB := FALSE;
	//Fehlerstruktur vorausfüllen
	stError.ObjectId := nObjectID;
	stError.HardwareGrp := E_HardwareGrp.Nothing;
	stError.POU := E_POU.POU_FB_SubstHolder;	
END_IF

CASE eCurrentState OF
	E_MachineState.MACHINESTATE_Active:
		IF bCooling THEN
			A_Cooling();
			IF nStateA_Cooling = 80 THEN
				bCooling := FALSE;
				nStateA_Cooling := 0;
				eCurrentAction := E_Action.ACTION_Nothing;
				eCurrentState := E_MachineState.MACHINESTATE_Idle;
				bBusy := FALSE;
			END_IF
		END_IF
END_CASE

//Prozessdaten aktualisieren
stProcessData.nObjId := nObjectID;
stProcessData.n32Data[0] := BOOL_TO_DINT(bIsInit);
stProcessData.n32Data[1] := eCurrentState;
stProcessData.n32Data[2] := stError.ErrorId;
IF pHeaterRef > 0 THEN
	nTempActual := pHeaterRef^.P_nTempActual;
	stProcessData.n32Data[3] := BOOL_TO_DINT(pHeaterRef^.P_bHeatingOn);
	stProcessData.n32Data[4] := UINT_TO_DINT(pHeaterRef^.P_nTempActual);
	stProcessData.n32Data[7] := BOOL_TO_DINT(pHeaterRef^.P_bEdgeLightOn);	
END_IF
stProcessData.n32Data[5] := BOOL_TO_DINT(aValves[nValveNrCool].bDigiOut1); 
stProcessData.n32Data[6] := BOOL_TO_DINT(bVacuumOk);

aObjProcData[nNotifyId] := stProcessData;

ACTION A_Cooling:
CASE nStateA_Cooling OF
	0:	aValves[nValveNrCool].M_On(1);
		nStateA_Cooling := 1;
		
	1:	//Warten bis Temp erreicht
		IF nTempActual <= nTempCooling THEN
			aValves[nValveNrCool].M_Off();
			nStateA_Cooling := 80;
		END_IF
		
		(*timerCooling(IN:= TRUE, PT:= T#2S);
		
		IF timerCooling.Q THEN
			timerCooling(IN:= FALSE);
			aValves[nValveNrCool].M_Off();
			nStateA_Cooling := 80;	
		END_IF*)
		
	70:	//Abbrechen
		aValves[nValveNrCool].M_Off();
		//timerCooling(IN:= FALSE);
		nStateA_Cooling := 80;
	
END_CASE
END_ACTION

METHOD FB_init : BOOL
VAR_INPUT
	bInitRetains : BOOL; // if TRUE, the retain variables are initialized (warm start / cold start)
	bInCopyCode : BOOL;  // if TRUE, the instance afterwards gets moved into the copy code (online change)
END_VAR
eObjectType := E_ObjectType.OBJECTTYPE_SubstHolder;
eObjectGroup := E_ObjectGroup.OBJECTGROUP_Target OR E_ObjectGroup.OBJECTGROUP_Device;
END_METHOD

METHOD M_AddChild : ERRORID
VAR_INPUT
	pObject : POINTER TO FB_Object;
	nSlotNr	: UINT;
	nIndex 	: INT;	
END_VAR

VAR
	pSlot : POINTER TO FB_Slot;
END_VAR
//In den abgeleiteten Tool-FBs wird überprüft, ob das entsprechende Objekt als Child tauglich ist
IF pObject > 0 THEN
	IF nSlotNr > 0 THEN
		pSlot := fbSlotList.M_GetAtNr(nSlotNr);
		IF pSlot > 0 THEN
			IF pSlot^.P_pChild = 0 THEN
				//Object darf selber noch an keinem Parent hängen
				IF pObject^.P_pParentObject = 0 THEN
					pSlot^.P_pChild := pObject;
					pObject^.P_pObjCollectNode := pObjCollectNode^.nodes.M_AddNewNode(pObject,nIndex);
					pObject^.M_UpdateParent();
				ELSE
					M_AddChild := E_ErrorIdObjMgmt.ERRORID_ObjectAlreadyOnAnotherParent;
				END_IF
			ELSE //Slot bereits belegt
				M_AddChild := E_ErrorIdObjMgmt.ERRORID_SlotIsAlreadyOccupied;
			END_IF		
		ELSE
			M_AddChild := E_ErrorIdObjMgmt.ERRORID_InvalidSlotNumber;			
		END_IF	
	ELSE
		M_AddChild := SUPER^.M_AddChild(pObject,nSlotNr,nIndex);
	END_IF
ELSE
	M_AddChild := E_ErrorIdObjMgmt.ERRORID_InvalidParentObject;
END_IF
END_METHOD

METHOD M_CancelAction
VAR_INPUT
	eAction : E_Action;
END_VAR
IF eAction = E_Action.ACTION_Cooling THEN
	IF bCooling AND nStateA_Cooling < 70 THEN
		nStateA_Cooling := 70;
	END_IF
END_IF
END_METHOD

METHOD M_CheckAction : ERRORID
VAR_INPUT
	refActionData	: REFERENCE TO ST_ActionData;
	pCorrelObject	: POINTER TO FB_Object;
END_VAR
IF NOT refActionData.eAction = E_Action.ACTION_MoveToTarget THEN
	M_CheckAction := E_ErrorIdCmd.ERRORID_InvalidAction;	
END_IF
END_METHOD

METHOD M_CheckProcDataType : BOOL
VAR_INPUT
	eProcDataType : E_ProcDataType;
END_VAR
IF eProcDataType = E_ProcDataType.PROCDATATYPE_Temp1 THEN
	M_CheckProcDataType := TRUE;
END_IF
END_METHOD

METHOD M_ClearAllProps
VAR_INPUT
	bIgnoreParent : BOOL; //Es wird das gesamte OD gelöscht. -> Zeiger auf Parent nicht mehr gültig!
END_VAR
fbSlotList.M_Reset();
SUPER^.M_ClearAllProps(bIgnoreParent);
END_METHOD

METHOD M_ExeAction : ERRORID
VAR_INPUT
	refActionData : REFERENCE TO ST_ActionData;
END_VAR
CASE refActionData.eAction OF
	E_Action.ACTION_Init:
		bIsInit := TRUE;
	E_Action.ACTION_Heating:	//Heizung ON/OFF
		IF pHeaterRef > 0 THEN
			nTempHeating := DINT_TO_USINT(refActionData.aParams[1]/10);
			bHeaterOn := DINT_TO_BOOL(refActionData.aParams[2]);	//Heizung "EIN"
			IF bHeaterOn THEN
				IF bCooling THEN
					nStateA_Cooling := 70;
				END_IF
				//aValves[nValveNrCool].M_Off();	//Kühlung "AUS"
				IF nTempHeating > 170 THEN
					M_ExeAction := E_ErrorIdCmd.ERRORID_InvalidHeatingTemp;
					RETURN;
				END_IF		
				pHeaterRef^.P_nTempSetpoint := nTempHeating;
				pHeaterRef^.P_bHeatingOn := TRUE;
			ELSE
				pHeaterRef^.P_bHeatingOn := FALSE;
			END_IF
		END_IF
	
	E_Action.ACTION_Cooling:	//Kühlung ON/OFF
		nTempCooling := DINT_TO_UINT(refActionData.aParams[1]);
		bCoolingOn := DINT_TO_BOOL(refActionData.aParams[2]);
		IF bCoolingOn THEN
			IF nValveNrCool = 0 THEN
				M_ExeAction := E_ErrorIdCmd.ERRORID_InvalidAction;
				RETURN;
			END_IF
			aValves[nValveNrCool].M_On(1); //Kühlung "EIN"
			IF pHeaterRef > 0 THEN
				pHeaterRef^.P_bHeatingOn := FALSE;	//Heizung "AUS"	
			END_IF
			
			bCooling := TRUE;
			eCurrentState := E_MachineState.MACHINESTATE_Active;
			eCurrentAction := E_Action.ACTION_Cooling;
			bBusy := TRUE;
		ELSE
			IF bCooling THEN
				nStateA_Cooling := 70;
			ELSE
				aValves[nValveNrCool].M_Off(); //Kühlung "AUS"	
			END_IF
		END_IF
		
	E_Action.ACTION_SwitchLight:	//Seitenlicht ON/OFF
		IF pHeaterRef > 0 THEN
			pHeaterRef^.P_bEdgeLightOn := DINT_TO_BOOL(refActionData.aParams[1]);	
		END_IF
		RETURN;
		
	E_Action.ACTION_SwitchPressure:
		IF refActionData.aParams[1] = 0 THEN
			aValves[nValveNrVac].M_Off();
			bVacuumOk := FALSE;
		ELSE
			aValves[nValveNrVac].M_On(1);
			bVacuumOk := TRUE;
		END_IF
	ELSE
		M_ExeAction := E_ErrorIdCmd.ERRORID_InvalidAction;
END_CASE
END_METHOD

METHOD M_GetAbsPos : ST_3DPoint
VAR_INPUT
	pChildPos	: POINTER TO ST_3DPoint;
	eTargetRef 	: E_TargetRef;
	nParam1		: UINT;
 	nParam2		: UINT;
	nParam3		: USINT;
	nParam4		: USINT;
	nZLevel		: USINT;
END_VAR
VAR_OUTPUT
	nErrorId 	: ERRORID;
	lrAngle		: LREAL;
END_VAR
VAR
	stLocPos : ST_3DPoint;
	pSlot : POINTER TO FB_Slot;
END_VAR
IF eTargetRef = E_TargetRef.TARGETREF_Slot THEN
	//Slotnummer checken
	pSlot := M_GetSlot(nParam1);
	IF pSlot > 0 THEN
		stLocPos := F_Add3DPoints(pSlot^.P_stRelPos,stRelPos);
		stLocPos.Z := stLocPos.Z + stDimension.Height;
		//kann es mal sein, dass hier das ParentTarget = 0 ist?
		//ja -> bei der Workplate
		IF pChildPos > 0 THEN
			stLocPos := F_Add3DPoints(stLocPos,pChildPos^);
		END_IF
		IF pParentTarget > 0 THEN
			IF pParentSlot > 0 THEN
				M_GetAbsPos := pParentTarget^.M_GetAbsPos(pChildPos := ADR(stLocPos), eTargetRef:= E_TargetRef.TARGETREF_Slot,
															nParam1:= pParentSlot^.P_nNr,
															nParam2:= 0, nParam3:= 0, nParam4:= 0, nZLevel:= 0, lrAngle=> lrAngle,
															nErrorId=> nErrorId);		
			ELSE
				M_GetAbsPos := pParentTarget^.M_GetAbsPos(pChildPos := ADR(stLocPos), eTargetRef:= E_TargetRef.TARGETREF_LeftBottom,
																nParam1:= 0,
																nParam2:= 0, nParam3:= 0,nParam4:= 0, nZLevel:= 0,
																lrAngle => lrAngle, nErrorId=> nErrorId);
			END_IF
		ELSE
			M_GetAbsPos := stLocPos;
		END_IF		
	ELSE
		nErrorId := E_ErrorIdCmd.ERRORID_InvalidTargetSlot;
	END_IF
	
ELSE
	M_GetAbsPos := SUPER^.M_GetAbsPos(pChildPos := pChildPos, eTargetRef:= eTargetRef,
													nParam1:= nParam1,
													nParam2:= nParam2, nParam3:= nParam3, nParam4:= 0, nZLevel:= nZLevel,
													lrAngle => lrAngle, nErrorId=> nErrorId);	
END_IF
END_METHOD

METHOD M_GetActionBusy : BOOL
VAR_INPUT
	eAction : E_Action;
END_VAR
M_GetActionBusy := (eCurrentAction = eAction);
END_METHOD

METHOD M_GetAllProps : ERRORID
VAR_INPUT
	refCmdData : REFERENCE TO  ST_CmdData;
END_VAR

VAR
	i : UINT;
	pSlot		: POINTER TO FB_Slot;
END_VAR
SUPER^.M_GetAllProps(refCmdData);

nCurrentPropIndex := nCurrentPropIndex + 1;

refCmdData.n32Data[nCurrentPropIndex] := fbSlotList.P_nCount;

fbSlotList.M_SetCurrentToHead();

FOR i := 1 TO fbSlotList.P_nCount BY 1 DO
	pSlot := fbSlotList.M_GetNext();
	IF pSlot > 0 THEN
		nCurrentPropIndex := nCurrentPropIndex + 1;
		refCmdData.n32Data[nCurrentPropIndex] := pSlot^.P_nNr;
		nCurrentPropIndex := nCurrentPropIndex + 1;
		refCmdData.n32Data[nCurrentPropIndex] := REAL_TO_DINT(pSlot^.P_rRelPosX);
		nCurrentPropIndex := nCurrentPropIndex + 1;
		refCmdData.n32Data[nCurrentPropIndex] := REAL_TO_DINT(pSlot^.P_rRelPosY);
		nCurrentPropIndex := nCurrentPropIndex + 1;
		refCmdData.n32Data[nCurrentPropIndex] := REAL_TO_DINT(pSlot^.P_rRelPosZ);
	END_IF		
END_FOR	

nCurrentPropIndex := nCurrentPropIndex + 1;
refCmdData.n32Data[nCurrentPropIndex] := nHeaterChannel;
IF pHeaterRef > 0 THEN
	nCurrentPropIndex := nCurrentPropIndex + 1;
	refCmdData.n32Data[nCurrentPropIndex] := pHeaterRef^.P_nPidKp;
	nCurrentPropIndex := nCurrentPropIndex + 1;
	refCmdData.n32Data[nCurrentPropIndex] := pHeaterRef^.P_nPidKi;
	nCurrentPropIndex := nCurrentPropIndex + 1;
	refCmdData.n32Data[nCurrentPropIndex] := pHeaterRef^.P_nPidKd;
	nCurrentPropIndex := nCurrentPropIndex + 1;
	refCmdData.n32Data[nCurrentPropIndex] := pHeaterRef^.P_nPidTa;
ELSE
	nCurrentPropIndex := nCurrentPropIndex + 1;
	refCmdData.n32Data[nCurrentPropIndex] := 0;
	nCurrentPropIndex := nCurrentPropIndex + 1;
	refCmdData.n32Data[nCurrentPropIndex] := 0;
	nCurrentPropIndex := nCurrentPropIndex + 1;
	refCmdData.n32Data[nCurrentPropIndex] := 0;
	nCurrentPropIndex := nCurrentPropIndex + 1;
	refCmdData.n32Data[nCurrentPropIndex] := 0;
END_IF
nCurrentPropIndex := nCurrentPropIndex + 1;
refCmdData.n32Data[nCurrentPropIndex] := nValveNrCool;
nCurrentPropIndex := nCurrentPropIndex + 1;
refCmdData.n32Data[nCurrentPropIndex] := nValveNrVac;
END_METHOD

METHOD M_GetProcData : DINT
VAR_INPUT
	eProcDataType : E_ProcDataType;
END_VAR
IF eProcDataType = E_ProcDataType.PROCDATATYPE_Temp1 THEN
	M_GetProcData := nTempActual;
END_IF
END_METHOD

METHOD M_GetSlot : POINTER TO FB_Slot
VAR_INPUT
	nSlotNr : UINT;
END_VAR
M_GetSlot := fbSlotList.M_GetAtNr(nSlotNr);
END_METHOD

METHOD M_GetSlotFromChild : POINTER TO FB_Slot
VAR_INPUT
	pObject : POINTER TO FB_Object;
END_VAR

VAR
	pSlot : POINTER TO FB_Slot;
END_VAR
//Die SlotList iterieren und vergleichen ob Objekte übereinstimmen
fbSlotList.M_SetCurrentToHead();
REPEAT
	pSlot := fbSlotList.M_GetNext();
	IF pSlot > 0 THEN
		IF pSlot^.P_pChild = pObject THEN
			M_GetSlotFromChild := pSlot;
			EXIT;
		END_IF
	END_IF
UNTIL pSlot = 0
END_REPEAT
END_METHOD

METHOD M_SetAllProps : ERRORID
VAR_INPUT
	refCmdData : REFERENCE TO  ST_CmdData;
END_VAR

VAR
	i : UINT;
	pSlot 		: POINTER TO FB_Slot;
END_VAR
M_SetAllProps := SUPER^.M_SetAllProps(refCmdData);

IF M_SetAllProps > 0 THEN
	RETURN;
END_IF

//Slots parametrieren
nCurrentPropIndex := nCurrentPropIndex + 1;
nFirstSlotPropIndex := nCurrentPropIndex;
nNumberOfSlots := DINT_TO_UINT(refCmdData.n32Data[nCurrentPropIndex]);

//Falls SlotList noch nicht existiert, dann neue erstellen
IF fbSlotList.P_nCount = 0 THEN
	FOR i:= 1 TO nNumberOfSlots BY 1 DO
		pSlot := __NEW(FB_Slot(pOwner := THIS));
		fbSlotList.M_Add(pSlot);
		nCurrentPropIndex := nCurrentPropIndex + 1;
		pSlot^.P_nNr := DINT_TO_USINT(refCmdData.n32Data[nCurrentPropIndex]);
		nCurrentPropIndex := nCurrentPropIndex + 1;
		pSlot^.P_rRelPosX := DINT_TO_REAL(refCmdData.n32Data[nCurrentPropIndex]);
		nCurrentPropIndex := nCurrentPropIndex + 1;
		pSlot^.P_rRelPosY := DINT_TO_REAL(refCmdData.n32Data[nCurrentPropIndex]);
		nCurrentPropIndex := nCurrentPropIndex + 1;
		pSlot^.P_rRelPosZ := DINT_TO_REAL(refCmdData.n32Data[nCurrentPropIndex]);
	END_FOR
ELSE
	IF nNumberOfSlots <> fbSlotList.P_nCount THEN	//Anzahl der Slots dürfen sich nicht ändern
		M_SetAllProps := E_ErrorIdObjMgmt.ERRORID_ChangeNoOfSlotsNotAllowed;
		RETURN;		
	END_IF

	FOR i:= 1 TO nNumberOfSlots BY 1 DO
		nCurrentPropIndex := nCurrentPropIndex + 1;
		pSlot := fbSlotList.M_GetAtNr(DINT_TO_USINT(refCmdData.n32Data[nCurrentPropIndex]));
		IF pSlot > 0 THEN
			nCurrentPropIndex := nCurrentPropIndex + 1;
			pSlot^.P_rRelPosX := DINT_TO_REAL(refCmdData.n32Data[nCurrentPropIndex]);
			nCurrentPropIndex := nCurrentPropIndex + 1;
			pSlot^.P_rRelPosY := DINT_TO_REAL(refCmdData.n32Data[nCurrentPropIndex]);
			nCurrentPropIndex := nCurrentPropIndex + 1;
			pSlot^.P_rRelPosZ := DINT_TO_REAL(refCmdData.n32Data[nCurrentPropIndex]);
		ELSE
			M_SetAllProps := 222;
			RETURN;
		END_IF	
	END_FOR
END_IF
nLastSlotPropIndex := nCurrentPropIndex;
nNoOfProps := nCurrentPropIndex + 1;

nCurrentPropIndex := nCurrentPropIndex + 1;
nSpecPropIndex := nCurrentPropIndex;
{IF defined (variable:afbSubstHeatRef)}
IF refCmdData.n32Data[nCurrentPropIndex] > 0 AND refCmdData.n32Data[nCurrentPropIndex] <= cNoOfSubstHeaters THEN
	nHeaterChannel := DINT_TO_USINT(refCmdData.n32Data[nCurrentPropIndex]);
	pHeaterRef := ADR(afbSubstHeatRef[nHeaterChannel]);
	nCurrentPropIndex := nCurrentPropIndex + 1;
	pHeaterRef^.P_nPidKp := DINT_TO_UINT(refCmdData.n32Data[nCurrentPropIndex]);
	nCurrentPropIndex := nCurrentPropIndex + 1;
	pHeaterRef^.P_nPidKi := DINT_TO_UINT(refCmdData.n32Data[nCurrentPropIndex]);
	nCurrentPropIndex := nCurrentPropIndex + 1;
	pHeaterRef^.P_nPidKd := DINT_TO_UINT(refCmdData.n32Data[nCurrentPropIndex]);
	nCurrentPropIndex := nCurrentPropIndex + 1;
	pHeaterRef^.P_nPidTa := DINT_TO_USINT(refCmdData.n32Data[nCurrentPropIndex]);
ELSIF refCmdData.n32Data[nCurrentPropIndex] = 0 THEN
	nHeaterChannel := 0;
	pHeaterRef := 0;
	nCurrentPropIndex := nCurrentPropIndex + 4;
ELSE
	M_SetAllProps := E_ErrorIdObjMgmt.ERRORID_InvalidHeaterChannel;
END_IF	
{ELSE}
M_SetAllProps := E_ErrorIdObjMgmt.ERRORID_InvalidHardwareRef;
{END_IF}
nCurrentPropIndex := nCurrentPropIndex + 1;
IF refCmdData.n32Data[nCurrentPropIndex] >= 0 AND refCmdData.n32Data[nCurrentPropIndex] <= cNoOfValves THEN
	nValveNrCool := DINT_TO_USINT(refCmdData.n32Data[nCurrentPropIndex]);
END_IF
nCurrentPropIndex := nCurrentPropIndex + 1;
IF refCmdData.n32Data[nCurrentPropIndex] > 0 AND refCmdData.n32Data[nCurrentPropIndex] <= cNoOfValves THEN
	nValveNrVac := DINT_TO_USINT(refCmdData.n32Data[nCurrentPropIndex]);	
END_IF

nNoOfProps := nCurrentPropIndex + 1;
END_METHOD

METHOD M_SetSingleProp : ERRORID
VAR_INPUT
	refCmdData : REFERENCE TO  ST_CmdData;
END_VAR
IF nSpecPropIndex = refCmdData.aHeader[1] THEN
	M_SetSingleProp := E_ErrorIdCmd.ERRORID_InvalidProperty; //HeaterChannel darf nicht verändert werden
ELSIF (nSpecPropIndex + 1) = refCmdData.aHeader[1] THEN
	IF pHeaterRef > 0 THEN
		pHeaterRef^.P_nPidKp := DINT_TO_UINT(refCmdData.n32Data[0]);
	ELSE
		M_SetSingleProp := E_ErrorIdCmd.ERRORID_InvalidProperty;
	END_IF	
ELSIF (nSpecPropIndex + 2) = refCmdData.aHeader[1] THEN
	IF pHeaterRef > 0 THEN
		pHeaterRef^.P_nPidKi := DINT_TO_UINT(refCmdData.n32Data[0]);
	ELSE
		M_SetSingleProp := E_ErrorIdCmd.ERRORID_InvalidProperty;
	END_IF	
ELSIF (nSpecPropIndex + 3) = refCmdData.aHeader[1] THEN
	IF pHeaterRef > 0 THEN
		pHeaterRef^.P_nPidKd := DINT_TO_UINT(refCmdData.n32Data[0]);
	ELSE
		M_SetSingleProp := E_ErrorIdCmd.ERRORID_InvalidProperty;
	END_IF	
ELSIF (nSpecPropIndex + 4) = refCmdData.aHeader[1] THEN
	IF pHeaterRef > 0 THEN
		pHeaterRef^.P_nPidTa := DINT_TO_USINT(refCmdData.n32Data[0]);
	ELSE
		M_SetSingleProp := E_ErrorIdCmd.ERRORID_InvalidProperty;
	END_IF	
ELSIF (nSpecPropIndex + 5) = refCmdData.aHeader[1] THEN
	IF refCmdData.n32Data[0] > 0 AND refCmdData.n32Data[0] <= cNoOfValves THEN
		nValveNrCool := DINT_TO_USINT(refCmdData.n32Data[0]);
	ELSE
		M_SetSingleProp := E_ErrorIdObjMgmt.ERRORID_InvalidValveNumber;
	END_IF	
ELSIF (nSpecPropIndex + 6) = refCmdData.aHeader[1] THEN
	IF refCmdData.n32Data[0] > 0 AND refCmdData.n32Data[0] <= cNoOfValves THEN
		nValveNrVac := DINT_TO_USINT(refCmdData.n32Data[0]);
	ELSE
		M_SetSingleProp := E_ErrorIdObjMgmt.ERRORID_InvalidValveNumber;
	END_IF	
ELSE
	M_SetSingleProp := SUPER^.M_SetSingleProp(refCmdData);
END_IF
END_METHOD

METHOD M_Stop : ERRORID
VAR_INPUT
END_VAR
IF bCooling THEN
	nStateA_Cooling := 70;
END_IF
END_METHOD

END_FUNCTION_BLOCK

// ---- Objects/Targets/Active/FB_SubstHolderUnistat.TcPOU
FUNCTION_BLOCK FB_SubstHolderUnistat EXTENDS FB_ActiveTarget IMPLEMENTS I_SlotTarget

VAR
	fbSlotList			: FB_SlotList;
	nNumberOfSlots		: UINT;
	nFirstSlotPropIndex	: UINT;	//erster Index für Slots (benötigt in M_SetSingleProps)
	nLastSlotPropIndex	: UINT;	//letzte Index für Slots (benötigt in M_SetSingleProps)

	//Hardware-Verküpfung
	//erfolgt direkt über die seriell Schnittstelle

	//Prozessdaten
	bVacuumOk			: BOOL;
	
	
	nCurrentTempIntern	: DINT;
	nCurrentTempExtern	: DINT;
	bTempControlIsOn	: BOOL;

	//Spec-Properties
	nValveNrVac			: USINT;	//VentilNr Vakuum (FBox)
	
	//****************************************Aktionvariablen****************************************************
	//Action: "TempControl"
	bTempControl		: BOOL;
	nTempSetpoint		: DINT; //1/10tel °C
	bTempControlOn		: BOOL;
	fbTempControl		: FB_UnistatControl;
	
END_VAR

IF bInitFB THEN
	bInitFB := FALSE;
	//Fehlerstruktur vorausfüllen
	stError.ObjectId := nObjectID;
	stError.HardwareGrp := E_HardwareGrp.Nothing;
	stError.POU := E_POU.POU_FB_SubstHolder;
END_IF

IF eCurrentState = E_MachineState.MACHINESTATE_Active THEN
	IF eCurrentAction = E_ACtion.ACTION_Cooling THEN
		fbTempControl(UnistatRef:= fbUnistatRef, nTempSetpoint:= nTempSetpoint, bTempControlOn:= bTempControlOn, bExecute:= TRUE);
		IF NOT fbTempControl.bBusy THEN
			IF fbTempControl.bError THEN
				//hier könnte man den Fehler melden?
			END_IF
			fbTempControl(bExecute:= FALSE);
			eCurrentAction := E_Action.ACTION_Nothing;
			eCurrentState := E_MachineState.MACHINESTATE_Idle;
			bBusy := FALSE;
		END_IF
	END_IF
END_IF

//Prozessdaten aktualisieren
stProcessData.nObjId := nObjectID;
stProcessData.n32Data[0] := BOOL_TO_DINT(bIsInit);
stProcessData.n32Data[1] := eCurrentState;
stProcessData.n32Data[2] := stError.ErrorId;

{IF defined(variable:fbUnistatRef)}
stProcessData.n32Data[3] := fbUnistatRef.P_eState;
nCurrentTempIntern := fbUnistatRef.P_nCurrentTempIntern;
stProcessData.n32Data[4] := nCurrentTempIntern;
nCurrentTempExtern := fbUnistatRef.P_nCurrentTempExtern;
stProcessData.n32Data[5] := nCurrentTempExtern;
{END_IF}
stProcessData.n32Data[6] := BOOL_TO_DINT(bVacuumOk);

aObjProcData[nNotifyId] := stProcessData;

METHOD FB_init : BOOL
VAR_INPUT
	bInitRetains : BOOL; // if TRUE, the retain variables are initialized (warm start / cold start)
	bInCopyCode : BOOL;  // if TRUE, the instance afterwards gets moved into the copy code (online change)
END_VAR
eObjectType := E_ObjectType.OBJECTTYPE_SubstHolderUnistat;
eObjectGroup := E_ObjectGroup.OBJECTGROUP_Target OR E_ObjectGroup.OBJECTGROUP_Device;
END_METHOD

METHOD M_AddChild : ERRORID
VAR_INPUT
	pObject : POINTER TO FB_Object;
	nSlotNr	: UINT;
	nIndex 	: INT;	
END_VAR

VAR
	pSlot : POINTER TO FB_Slot;
END_VAR
//In den abgeleiteten Tool-FBs wird überprüft, ob das entsprechende Objekt als Child tauglich ist
IF pObject > 0 THEN
	IF nSlotNr > 0 THEN
		pSlot := fbSlotList.M_GetAtNr(nSlotNr);
		IF pSlot > 0 THEN
			IF pSlot^.P_pChild = 0 THEN
				//Object darf selber noch an keinem Parent hängen
				IF pObject^.P_pParentObject = 0 THEN
					pSlot^.P_pChild := pObject;
					pObject^.P_pObjCollectNode := pObjCollectNode^.nodes.M_AddNewNode(pObject,nIndex);
					pObject^.M_UpdateParent();
				ELSE
					M_AddChild := E_ErrorIdObjMgmt.ERRORID_ObjectAlreadyOnAnotherParent;
				END_IF
			ELSE //Slot bereits belegt
				M_AddChild := E_ErrorIdObjMgmt.ERRORID_SlotIsAlreadyOccupied;
			END_IF		
		ELSE
			M_AddChild := E_ErrorIdObjMgmt.ERRORID_InvalidSlotNumber;			
		END_IF	
	ELSE
		M_AddChild := SUPER^.M_AddChild(pObject,nSlotNr,nIndex);
	END_IF
ELSE
	M_AddChild := E_ErrorIdObjMgmt.ERRORID_InvalidParentObject;
END_IF
END_METHOD

METHOD M_CheckAction : ERRORID
VAR_INPUT
	refActionData	: REFERENCE TO ST_ActionData;
	pCorrelObject	: POINTER TO FB_Object;
END_VAR
IF NOT refActionData.eAction = E_Action.ACTION_MoveToTarget THEN
	M_CheckAction := E_ErrorIdCmd.ERRORID_InvalidAction;	
END_IF
END_METHOD

METHOD M_CheckProcDataType : BOOL
VAR_INPUT
	eProcDataType : E_ProcDataType;
END_VAR
IF eProcDataType = E_ProcDataType.PROCDATATYPE_Temp1 OR eProcDataType = E_ProcDataType.PROCDATATYPE_Temp2 THEN
	M_CheckProcDataType := TRUE;
END_IF
END_METHOD

METHOD M_ClearAllProps
VAR_INPUT
	bIgnoreParent : BOOL; //Es wird das gesamte OD gelöscht. -> Zeiger auf Parent nicht mehr gültig!
END_VAR
fbSlotList.M_Reset();
SUPER^.M_ClearAllProps(bIgnoreParent);
END_METHOD

METHOD M_ExeAction : ERRORID
VAR_INPUT
	refActionData : REFERENCE TO ST_ActionData;
END_VAR
CASE refActionData.eAction OF
	E_Action.ACTION_Init:
		bIsInit := TRUE;
	
	E_Action.ACTION_Cooling:	//Temperierung on/off
		nTempSetpoint := refActionData.aParams[1];
		bTempControlOn := DINT_TO_BOOL(refActionData.aParams[2]);
		eCurrentState := E_MachineState.MACHINESTATE_Active;
		eCurrentAction := E_Action.ACTION_Cooling;
		bBusy := TRUE;
		
	E_Action.ACTION_SwitchPressure:
		IF refActionData.aParams[1] = 0 THEN
			aValves[nValveNrVac].M_Off();
			bVacuumOk := FALSE;
		ELSE
			aValves[nValveNrVac].M_On(1);
			bVacuumOk := TRUE;
		END_IF
	ELSE
		M_ExeAction := E_ErrorIdCmd.ERRORID_InvalidAction;
END_CASE
END_METHOD

METHOD M_GetAbsPos : ST_3DPoint
VAR_INPUT
	pChildPos	: POINTER TO ST_3DPoint;
	eTargetRef 	: E_TargetRef;
	nParam1		: UINT;
 	nParam2		: UINT;
	nParam3		: USINT;
	nZLevel		: USINT;
END_VAR
VAR_OUTPUT
	nErrorId 	: ERRORID;
	lrAngle		: LREAL;
END_VAR
VAR
	stLocPos : ST_3DPoint;
	pSlot : POINTER TO FB_Slot;
END_VAR
IF eTargetRef = E_TargetRef.TARGETREF_Slot THEN
	//Slotnummer checken
	pSlot := M_GetSlot(nParam1);
	IF pSlot > 0 THEN
		stLocPos := F_Add3DPoints(pSlot^.P_stRelPos,stRelPos);
		stLocPos.Z := stLocPos.Z + stDimension.Height;
		//kann es mal sein, dass hier das ParentTarget = 0 ist?
		//ja -> bei der Workplate
		IF pChildPos > 0 THEN
			stLocPos := F_Add3DPoints(stLocPos,pChildPos^);
		END_IF
		IF pParentTarget > 0 THEN
			IF pParentSlot > 0 THEN
				M_GetAbsPos := pParentTarget^.M_GetAbsPos(pChildPos := ADR(stLocPos), eTargetRef:= E_TargetRef.TARGETREF_Slot,
															nParam1:= pParentSlot^.P_nNr,
															nParam2:= 0, nParam3:= 0,nZLevel:= 0, lrAngle=> lrAngle,
															nErrorId=> nErrorId);		
			ELSE
				M_GetAbsPos := pParentTarget^.M_GetAbsPos(pChildPos := ADR(stLocPos), eTargetRef:= E_TargetRef.TARGETREF_LeftBottom,
																nParam1:= 0,
																nParam2:= 0, nParam3:= 0,nZLevel:= 0,
																lrAngle => lrAngle, nErrorId=> nErrorId);
			END_IF
		ELSE
			M_GetAbsPos := stLocPos;
		END_IF		
	ELSE
		nErrorId := E_ErrorIdCmd.ERRORID_InvalidTargetSlot;
	END_IF
	
ELSE
	M_GetAbsPos := SUPER^.M_GetAbsPos(pChildPos := pChildPos, eTargetRef:= eTargetRef,
													nParam1:= nParam1,
													nParam2:= nParam2, nParam3:= nParam3, nZLevel:= nZLevel,
													lrAngle => lrAngle, nErrorId=> nErrorId);	
END_IF
END_METHOD

METHOD M_GetActionBusy : BOOL
VAR_INPUT
	eAction : E_Action;
END_VAR
M_GetActionBusy := (eCurrentAction = eAction);
END_METHOD

METHOD M_GetAllProps : ERRORID
VAR_INPUT
	refCmdData : REFERENCE TO  ST_CmdData;
END_VAR

VAR
	i : UINT;
	pSlot		: POINTER TO FB_Slot;
END_VAR
SUPER^.M_GetAllProps(refCmdData);

nCurrentPropIndex := nCurrentPropIndex + 1;

refCmdData.n32Data[nCurrentPropIndex] := fbSlotList.P_nCount;

fbSlotList.M_SetCurrentToHead();

FOR i := 1 TO fbSlotList.P_nCount BY 1 DO
	pSlot := fbSlotList.M_GetNext();
	IF pSlot > 0 THEN
		nCurrentPropIndex := nCurrentPropIndex + 1;
		refCmdData.n32Data[nCurrentPropIndex] := pSlot^.P_nNr;
		nCurrentPropIndex := nCurrentPropIndex + 1;
		refCmdData.n32Data[nCurrentPropIndex] := REAL_TO_DINT(pSlot^.P_rRelPosX);
		nCurrentPropIndex := nCurrentPropIndex + 1;
		refCmdData.n32Data[nCurrentPropIndex] := REAL_TO_DINT(pSlot^.P_rRelPosY);
		nCurrentPropIndex := nCurrentPropIndex + 1;
		refCmdData.n32Data[nCurrentPropIndex] := REAL_TO_DINT(pSlot^.P_rRelPosZ);
	END_IF		
END_FOR	

nCurrentPropIndex := nCurrentPropIndex + 1;
refCmdData.n32Data[nCurrentPropIndex] := nValveNrVac;
END_METHOD

METHOD M_GetProcData : DINT
VAR_INPUT
	eProcDataType : E_ProcDataType;
END_VAR
IF eProcDataType = E_ProcDataType.PROCDATATYPE_Temp1 THEN
	M_GetProcData := nCurrentTempIntern;
ELSIF eProcDataType = E_ProcDataType.PROCDATATYPE_Temp2 THEN
	M_GetProcData := nCurrentTempExtern;
END_IF
END_METHOD

METHOD M_GetSlot : POINTER TO FB_Slot
VAR_INPUT
	nSlotNr : UINT;
END_VAR
M_GetSlot := fbSlotList.M_GetAtNr(nSlotNr);
END_METHOD

METHOD M_GetSlotFromChild : POINTER TO FB_Slot
VAR_INPUT
	pObject : POINTER TO FB_Object;
END_VAR

VAR
	pSlot : POINTER TO FB_Slot;
END_VAR
//Die SlotList iterieren und vergleichen ob Objekte übereinstimmen
fbSlotList.M_SetCurrentToHead();
REPEAT
	pSlot := fbSlotList.M_GetNext();
	IF pSlot > 0 THEN
		IF pSlot^.P_pChild = pObject THEN
			M_GetSlotFromChild := pSlot;
			EXIT;
		END_IF
	END_IF
UNTIL pSlot = 0
END_REPEAT
END_METHOD

METHOD M_SetAllProps : ERRORID
VAR_INPUT
	refCmdData : REFERENCE TO  ST_CmdData;
END_VAR

VAR
	i : UINT;
	pSlot 		: POINTER TO FB_Slot;
END_VAR
M_SetAllProps := SUPER^.M_SetAllProps(refCmdData);

IF M_SetAllProps > 0 THEN
	RETURN;
END_IF

//Slots parametrieren
nCurrentPropIndex := nCurrentPropIndex + 1;
nFirstSlotPropIndex := nCurrentPropIndex;
nNumberOfSlots := DINT_TO_UINT(refCmdData.n32Data[nCurrentPropIndex]);

//Falls SlotList noch nicht existiert, dann neue erstellen
IF fbSlotList.P_nCount = 0 THEN
	FOR i:= 1 TO nNumberOfSlots BY 1 DO
		pSlot := __NEW(FB_Slot(pOwner := THIS));
		fbSlotList.M_Add(pSlot);
		nCurrentPropIndex := nCurrentPropIndex + 1;
		pSlot^.P_nNr := DINT_TO_USINT(refCmdData.n32Data[nCurrentPropIndex]);
		nCurrentPropIndex := nCurrentPropIndex + 1;
		pSlot^.P_rRelPosX := DINT_TO_REAL(refCmdData.n32Data[nCurrentPropIndex]);
		nCurrentPropIndex := nCurrentPropIndex + 1;
		pSlot^.P_rRelPosY := DINT_TO_REAL(refCmdData.n32Data[nCurrentPropIndex]);
		nCurrentPropIndex := nCurrentPropIndex + 1;
		pSlot^.P_rRelPosZ := DINT_TO_REAL(refCmdData.n32Data[nCurrentPropIndex]);
	END_FOR
ELSE
	IF nNumberOfSlots <> fbSlotList.P_nCount THEN	//Anzahl der Slots dürfen sich nicht ändern
		M_SetAllProps := E_ErrorIdObjMgmt.ERRORID_ChangeNoOfSlotsNotAllowed;
		RETURN;		
	END_IF

	FOR i:= 1 TO nNumberOfSlots BY 1 DO
		nCurrentPropIndex := nCurrentPropIndex + 1;
		pSlot := fbSlotList.M_GetAtNr(DINT_TO_USINT(refCmdData.n32Data[nCurrentPropIndex]));
		IF pSlot > 0 THEN
			nCurrentPropIndex := nCurrentPropIndex + 1;
			pSlot^.P_rRelPosX := DINT_TO_REAL(refCmdData.n32Data[nCurrentPropIndex]);
			nCurrentPropIndex := nCurrentPropIndex + 1;
			pSlot^.P_rRelPosY := DINT_TO_REAL(refCmdData.n32Data[nCurrentPropIndex]);
			nCurrentPropIndex := nCurrentPropIndex + 1;
			pSlot^.P_rRelPosZ := DINT_TO_REAL(refCmdData.n32Data[nCurrentPropIndex]);
		ELSE
			M_SetAllProps := 222;
			RETURN;
		END_IF	
	END_FOR
END_IF
nLastSlotPropIndex := nCurrentPropIndex;
nNoOfProps := nCurrentPropIndex + 1;

{IF NOT defined (variable:afbSubstHeatRef)}
	M_SetAllProps := E_ErrorIdObjMgmt.ERRORID_InvalidHardwareRef;
{END_IF}
nCurrentPropIndex := nCurrentPropIndex + 1;
IF refCmdData.n32Data[nCurrentPropIndex] > 0 AND refCmdData.n32Data[nCurrentPropIndex] <= cNoOfValves THEN
	nValveNrVac := DINT_TO_USINT(refCmdData.n32Data[nCurrentPropIndex]);	
END_IF

nNoOfProps := nCurrentPropIndex + 1;
END_METHOD

